			iStepSectionWork:=iStepSection;		(* set the actual section which is working *)
			IF ((iStepSection + (iStartSection - 1)) < iEndSection) THEN	(* check if the end section is active *)
				iStepSection:=iStepSection + 1;
			ELSE
				iStepSection:=5;	(* end section is reached-->go the displace procedure *)
			END_IF;
	(* plunge procedure *)
	5:		rActualPositionGrindFeedStart[5]:=rActualPositionGrindFeedEnd[iEndSection - (iStartSection - 1)];	(* set the new diameter of the section which will going to work *)
			rDistanceToWorkedTool:=rActualPositionGrindFeedStart[5] - rToolDiameterWithOffset;	(* check the distance to the end diameter, which will go to work *)
			rGrindingRelativePosition:=rDistanceToWorkedTool;
			IF (rActualPositionGrindFeedStart[5] = T_Geometry.arEndDiameter[iEndSection]) THEN
				axWorkEndSection[5]:=TRUE;		(* the end of this section is reached *)
			ELSE
				axWorkEndSection[5]:=FALSE;		(* the end of this section is not reached *)
			END_IF;
			rActualPositionGrindFeedEnd[5]:=rToolDiameterWithOffset;
			iStepSectionWork:=iStepSection;		(* set the actual section which is working *)
			iStepSection:=0;
END_CASE;
END_FUNCTION_BLOCK

(* POU PRG_VISU_LAYER5/FB_VISU/iFctGetEditParaList, ST *)
FUNCTION iFctGetEditParaList : INT
VAR_INPUT
	dwActualPage:DWORD;		(* activate page on the visualisation *)
	xMicroRodActive: BOOL;		(* choice of the machine MicroWire or MicroRod *)
	iSelectParaList:INT;			(* parameter list choiced on the QVis *)
	iSelectParaListTeachRot:INT;	(* parameter list choiced on the QVis for teach ToolRotation *)
END_VAR
VAR
	iTmpRetEditParaList: INT;
END_VAR
(****************************************************************************************************************************************************)
(***********          This Function check the state of the parameter level and give the number of the parameter list                ************)
(****************************************************************************************************************************************************)
iTmpRetEditParaList:=0;
CASE dwActualPage OF
	110:	IF xMicroRodActive THEN
			iTmpRetEditParaList:=111;
		ELSE
			iTmpRetEditParaList:=110;
		END_IF;
	120:	IF (iSelectParaList = 0) OR (iSelectParaList = 1) THEN
			IF xMicroRodActive THEN
				iTmpRetEditParaList:=123;
			ELSE
				iTmpRetEditParaList:=120;
			END_IF;
		END_IF;
		IF (iSelectParaList = 2) THEN
			iTmpRetEditParaList:=121;
		END_IF;
		IF (iSelectParaList = 3) THEN
			IF xMicroRodActive THEN
				iTmpRetEditParaList:=125;
			ELSE
				iTmpRetEditParaList:=122;
			END_IF;
		END_IF;
	130:	IF xMicroRodActive THEN
			iTmpRetEditParaList:=131;
		ELSE
			iTmpRetEditParaList:=130;
		END_IF;
	140:	iTmpRetEditParaList:=140;
	150:	iTmpRetEditParaList:=150;
	210:	IF (iSelectParaListTeachRot = 0) OR (iSelectParaListTeachRot = 1) THEN
			iTmpRetEditParaList:=210;
		END_IF;
		IF (iSelectParaListTeachRot = 2) THEN
			iTmpRetEditParaList:=211;
		END_IF;
		IF (iSelectParaListTeachRot = 3) THEN
			iTmpRetEditParaList:=212;
		END_IF;
	220:	iTmpRetEditParaList:=0;
	230:	iTmpRetEditParaList:=230;
	310:IF xMicroRodActive THEN
			iTmpRetEditParaList:=311;
		ELSE
			iTmpRetEditParaList:=310;
		END_IF;
	320:	iTmpRetEditParaList:=0;
	410:	iTmpRetEditParaList:=410;
	420:	iTmpRetEditParaList:=0;
	430:	iTmpRetEditParaList:=0;
END_CASE;
iFctGetEditParaList:=iTmpRetEditParaList;
END_FUNCTION

(* POU PRG_VISU_LAYER5/FB_VISU/iFctReturnConfMessage, ST *)
FUNCTION iFctReturnConfMessage : INT
VAR_INPUT
	iNumAction:INT;	(* number of called action on the visualisation *)
END_VAR
VAR
END_VAR
(****************************************************************************************************************************************************)
(***********                      This Function check the action on the visu and gives a correspond message number                     ************)
(****************************************************************************************************************************************************)
	CASE iNumAction OF
	(* Action exceeded Timeout *)
	-1:	iFctReturnConfMessage:=102;
	(* NovRAM, 'Parameter saved' with confirmation *)
	1005:	iFctReturnConfMessage:=1;
	(* NovRAM, 'Parameter saved' without confirmation *)
	1006:	iFctReturnConfMessage:=1;
	(* Reference machine done *)
	1110:	iFctReturnConfMessage:=23;
	(* Process machine done *)
	1150:	iFctReturnConfMessage:=21;
	(* Process station done *)
	1151..1153:	iFctReturnConfMessage:=22;
	(* change page, no message *)
	10001..10999:	iFctReturnConfMessage:=0;
	(* Info , 'Confirm action' *)
	ELSE	iFctReturnConfMessage:=2;
	END_CASE
END_FUNCTION

(* POU PRG_VISU_LAYER5/FB_VISU/xFctCtrleProfileName, ST *)
FUNCTION xFctCtrleProfileName : BOOL
VAR_INPUT
	sNewProfileName:STRING(30);		(* profile name to save *)
	ptrProfileList:POINTER TO ARRAY[1..csiMaxProfile] OF ST_PROFILE_ID;	(* list of the saved profil names *)
END_VAR
VAR
(* variable *)
	i: INT;
	sTmp:STRING;
	sTmp2:STRING;
END_VAR
(****************************************************************************************************************************************************)
(***********                                              This Function check the name of the profile if it is correct                                                     ************)
(****************************************************************************************************************************************************)
(* Init. function *)
	xFctCtrleProfileName:=FALSE;
	sTmp:=FCT_UPLOW_CASE(	xLowConvert:=TRUE,
							sInString:=sNewProfileName);

(* Search if name already exists *)
	FOR i:=1 TO csiMaxProfile DO
		sTmp2:=	FCT_UPLOW_CASE(	xLowConvert:=TRUE,
								sInString:=ptrProfileList^[i].sName);
		IF sTmp = sTmp2 AND sTmp2 <> '' THEN RETURN; END_IF
	END_FOR

(* Confirm function *)
	xFctCtrleProfileName:=TRUE;
END_FUNCTION

(* POU GENERAL/FCT_UPLOW_CASE, ST *)
FUNCTION FCT_UPLOW_CASE : STRING
VAR_INPUT
	xLowConvert:BOOL;			(* FALSE=conversion to up case, TRUE=conversion in low case *)
	sInString:STRING;				(* string with 80 character, which will be convert *)
END_VAR
VAR
(* variable *)
	sListUpCase:STRING:='ABCDEFGHIJKLMNOPQRSTUVWXYZ';
	sListLowCase:STRING:='abcdefghijklmnopqrstuvwxyz';
	i:INT;
(* Tmp *)
	sTmp:STRING;
	iTmp:INT;
END_VAR
(****************************************************************************************************************************************************)
(***********                                                      This function convert a String in up or low case                                                                ************)
(****************************************************************************************************************************************************)
(* Init. *)
	FCT_UPLOW_CASE:='';

(*Test string size*)
	IF LEN(sInString) < 1 OR LEN(sInString) > 255 THEN RETURN; END_IF

	IF xLowConvert THEN
	(* Conversion to low case *)
		FOR i:= 1 TO LEN(sInString) DO
			sTmp:=MID(sInString,1,i);
			iTmp:=FIND(sListUpCase,sTmp);
			IF iTmp > 0 THEN FCT_UPLOW_CASE:=CONCAT(FCT_UPLOW_CASE,MID(sListLowCase,1,iTmp));
				ELSE FCT_UPLOW_CASE:=CONCAT(FCT_UPLOW_CASE,sTmp); END_IF
		END_FOR
	(* Conversion to up case *)
	ELSE
		FOR i:= 1 TO LEN(sInString) DO
			sTmp:=MID(sInString,1,i);
			iTmp:=FIND(sListLowCase,sTmp);
			IF iTmp > 0 THEN FCT_UPLOW_CASE:=CONCAT(FCT_UPLOW_CASE,MID(sListUpCase,1,iTmp));
				ELSE FCT_UPLOW_CASE:=CONCAT(FCT_UPLOW_CASE,sTmp); END_IF
		END_FOR
	END_IF
END_FUNCTION

(* POU PRG_VISU_LAYER5/FB_VISU/iFctExistProfileName, ST *)
FUNCTION iFctExistProfileName : INT
VAR_INPUT
	sProfileName:STRING(30);											(* name of the profile, which will be saved *)
	ptrProfileList:POINTER TO ARRAY[1..csiMaxProfile] OF ST_PROFILE_ID;	(* list of profil names which are saved *)
END_VAR
VAR
	i:INT;
	sTmp:STRING;
	sTmp2:STRING;
END_VAR
(****************************************************************************************************************************************************)
(***********                                               This Function check if the name of the profile already exists                                              ************)
(****************************************************************************************************************************************************)
(* Init. function *)
	iFctExistProfileName:=0;
	sTmp:=FCT_UPLOW_CASE(	xLowConvert:=TRUE,
							sInString:=sProfileName);

(* Search if name already exists *)
	FOR i:=1 TO csiMaxProfile DO
		sTmp2:=	FCT_UPLOW_CASE(	xLowConvert:=TRUE,
								sInString:=ptrProfileList^[i].sName);
		IF sTmp = sTmp2 AND sTmp2 <> '' THEN iFctExistProfileName:=i; RETURN; END_IF
	END_FOR
END_FUNCTION

(* POU PRG_VISU_LAYER5/FB_VISU/rFctCalcMaxToolDiameter, ST *)
FUNCTION rFctCalcMaxToolDiameter : REAL
VAR_INPUT
	rDistanceD1:REAL;		(* distance d1 of the prisma *)
	rDistanceD2:REAL;		(* distance d2 of the prisma *)
	rAnglePrism:REAL;		(* angle of the prisma *)
END_VAR
VAR
	rTmp: REAL;
	rTmpMaxDia: REAL;
END_VAR
(****************************************************************************************************************************************************)
(***********                    This Function calculate the maximum of the tooldiameter in case of the settled prisma                      ************)
(****************************************************************************************************************************************************)
rTmp:=SIN((90 - rAnglePrism/2) * PI/180);
IF rTmp <> 0 THEN
	rTmpMaxDia:=rDistanceD1/rTmp;
ELSE
	rTmpMaxDia:=0;
END_IF;
rFctCalcMaxToolDiameter:=rTmpMaxDia;
END_FUNCTION

(* POU PRG_VISU_LAYER5/FB_VISU/rFctCalcMinToolDiameter, ST *)
FUNCTION rFctCalcMinToolDiameter : REAL
VAR_INPUT
	rDistanceD1:REAL;		(* distance d1 of the prisma *)
	rDistanceD2:REAL;		(* distance d2 of the prisma *)
	rAnglePrism:REAL;		(* angle of the prisma *)
	bStateInputPrisma:BYTE;	(* choice of selected prisma *)
END_VAR
VAR
	rTmp: REAL;
	rTmp1: REAL;
	rMinD1_1: REAL;
	rMinD1_2: REAL;
	rReturnValue: REAL;
END_VAR
(****************************************************************************************************************************************************)
(***********                    This Function calculate the minimum of the tooldiameter in case of the settled prisma                      ************)
(****************************************************************************************************************************************************)
rFctCalcMinToolDiameter:=0;
rTmp:=TAN((rAnglePrism/2)*PI/180);
rTmp1:=SIN((rAnglePrism/2)*PI/180);
IF (rTmp <> 0) AND (rTmp1 <> 0) THEN
	rMinD1_1:=rDistanceD1/(rTmp * (1 + 1/rTmp1));
END_IF;
rMinD1_2:=rDistanceD2;
IF (bStateInputPrisma = 0) OR (bStateInputPrisma = 1) THEN
	IF (rMinD1_1 >= rMinD1_2) THEN
		rReturnValue:=rMinD1_1;
	ELSE
		rReturnValue:=rMinD1_2;
	END_IF;
ELSE
	rReturnValue:=rMinD1_1;
END_IF;
rFctCalcMinToolDiameter:=rReturnValue;
END_FUNCTION

(* POU PRG_VISU_LAYER5/FB_VISU/rFctCalcPrismaFactor, ST *)
FUNCTION rFctCalcPrismaFactor : REAL
VAR_INPUT
	rAnglePrism:REAL;	(* angle of the prisma *)
END_VAR
VAR
	rFactorPrisma: REAL;
END_VAR
(****************************************************************************************************************************************************)
(***********     This Function calculate the correctur factor for the GrindFeeder Axis dependent of the settled prisma         ************)
(****************************************************************************************************************************************************)
rFctCalcPrismaFactor:=0.0;
rFactorPrisma:=(1 + SIN((rAnglePrism / 2.0) * PI/180)) / (2.0 * SIN((rAnglePrism / 2.0) * PI / 180.0));
(* Auf 5 Kommastellen runden *)
rFactorPrisma:=	STRING_TO_REAL(	LREAL_TO_FMTSTR(	in:=rFactorPrisma,
														iPrecision:=5,
														bRound:=TRUE));

rFctCalcPrismaFactor:=rFactorPrisma;
END_FUNCTION

(* POU PRG_VISU_LAYER5/FB_VISU/FB_CTRLEBUTTON, ST *)
FUNCTION_BLOCK FB_CTRLEBUTTON
VAR_INPUT
	xHWStart:BOOL;							(* external start button *)
	xHWStop:BOOL;							(* external stop button *)
	dwActualPage:DWORD;					(* active number page of the visualisation *)
	T_VisuQVis:ST_QVIS;						(* data structure of the visualisation *)
	T_ExchgParam:ST_QVIS_EXCHG_PARAM;	(* data structure of the visualisation *)
	IxSafetyCircuitOn1:BOOL;					(* state of current if it is on or off from the channel 1 *)
	IxSafetyCircuitOn2:BOOL;					(* state of current if it is on or off from the channel 2 *)
END_VAR
VAR_OUTPUT
END_VAR
VAR_IN_OUT
	T_StartButton: ST_BUTTON;				(* data structure of the control button start *)
	T_StopButton:ST_BUTTON;				(* data structure of the control button stop *)
END_VAR
VAR
(* Init. variable *)
	xFirstExecution:BOOL:=FALSE;
(* Variable *)
	iIndexActivPage:INT;
	dwOldActualPage:DWORD;
(* FB Mask *)
	xMaskPageBtStart:BOOL;
	xMaskPageBtStop:BOOL;
(* Trigger *)
	RisingEdgeSignalStartButton:R_TRIG;
	RisingEdgeStartState:R_TRIG;
	RisingEdgeCfgBtStart:R_TRIG;
	RisingEdgeSignalStopButton:R_TRIG;
	RisingEdgeFlagStopProcess:R_TRIG;
(* Tmp variable *)
	xTmp:BOOL;
END_VAR
(****************************************************************************************************************************************************)
(***********             This Functionblock manage the external start and stop butto, also for the lamp of this button                  ************)
(****************************************************************************************************************************************************)
(* First execution *)
	IF NOT xFirstExecution THEN
		dwOldActualPage:=16#FFFFFFFF;
		RisingEdgeSignalStartButton(CLK:=FALSE);
		RisingEdgeStartState(CLK:=FALSE);
		RisingEdgeCfgBtStart(CLK:=FALSE);
		RisingEdgeSignalStopButton(CLK:=FALSE);
		RisingEdgeFlagStopProcess(CLK:=FALSE);
		(* Set first execution *)
		xFirstExecution:=TRUE;
	END_IF

(* exit FB if Qvis inactiv *)
	IF NOT(T_VisuQVis.T_CtrleVisu.xQvis) THEN RETURN; END_IF
	IF (dwActualPage < 1) OR (dwActualPage > 999) THEN RETURN; END_IF;

(* Index Activ Page *)
	IF dwActualPage = 0 THEN iIndexActivPage:=1;
	ELSE iIndexActivPage:=T_VisuQVis.T_PageIndex[dwActualPage].iIndexConfigPage; END_IF

(* Start Button *)
	xMaskPageBtStart:=FALSE;
	CASE dwActualPage OF
	(* Auto Geometry page *)
	10:	xTmp:=TRUE;
		IF xTmp AND (NOT(IxSafetyCircuitOn1) OR NOT(IxSafetyCircuitOn2)) THEN
			xTmp:=FALSE;	(* Energieversorgung muss eingeschaltet sein *)
		END_IF;
		IF xTmp AND ((T_ExchgParam.T_SafetyCtrl.bStateMessageError <> 0) OR (T_ExchgParam.T_SafetyCtrl.bStateMessageInfo <> 0)) THEN
			xTmp:=FALSE;
		END_IF;
		IF (T_ExchgParam.T_Visu.T_Message.iState = 401) OR (T_ExchgParam.T_Visu.T_Message.iState = 118) OR (T_ExchgParam.T_Visu.T_Message.iState = 119) OR (T_ExchgParam.T_Visu.T_Message.iState = 108) THEN
			xTmp:=FALSE;
		END_IF;
		(* copy state *)
		xMaskPageBtStart:=xTmp;
	(* Auto Groove page *)
	20:	xTmp:=TRUE;
		IF xTmp AND (NOT(IxSafetyCircuitOn1) OR NOT(IxSafetyCircuitOn2)) THEN
			xTmp:=FALSE;	(* Energieversorgung muss eingeschaltet sein *)
		END_IF;
		IF xTmp AND ((T_ExchgParam.T_SafetyCtrl.bStateMessageError <> 0) OR (T_ExchgParam.T_SafetyCtrl.bStateMessageInfo <> 0)) THEN
			xTmp:=FALSE;
		END_IF;
		IF (T_ExchgParam.T_Visu.T_Message.iState = 401) OR (T_ExchgParam.T_Visu.T_Message.iState = 118) OR (T_ExchgParam.T_Visu.T_Message.iState = 119) OR (T_ExchgParam.T_Visu.T_Message.iState = 108) THEN
			xTmp:=FALSE;
		END_IF;
		(* copy state *)
		xMaskPageBtStart:=xTmp;
	(* Reference page *)
	30:	xTmp:=TRUE;
		IF xTmp AND (NOT(IxSafetyCircuitOn1) OR NOT(IxSafetyCircuitOn2)) THEN
			xTmp:=FALSE;	(* Energieversorgung muss eingeschaltet sein *)
		END_IF;
		IF xTmp AND ((T_ExchgParam.T_SafetyCtrl.bStateMessageError <> 0) OR (T_ExchgParam.T_SafetyCtrl.bStateMessageInfo <> 0)) THEN
			xTmp:=FALSE;
		END_IF;
		IF (T_ExchgParam.T_Visu.T_Message.iState = 401) OR (T_ExchgParam.T_Visu.T_Message.iState = 118) OR (T_ExchgParam.T_Visu.T_Message.iState = 119) THEN
			xTmp:=FALSE;
		END_IF;
		IF (T_ExchgParam.T_StationCommon.iConfigMachineType = 1) THEN
			xTmp:=FALSE;
		END_IF;
		(* copy state *)
		xMaskPageBtStart:=xTmp;
	(* Tool Calibration page *)
	110:	xTmp:=TRUE;
		IF xTmp AND (NOT(IxSafetyCircuitOn1) OR NOT(IxSafetyCircuitOn2)) THEN
			xTmp:=FALSE;	(* Energieversorgung muss eingeschaltet sein *)
		END_IF;
		IF xTmp AND ((T_ExchgParam.T_SafetyCtrl.bStateMessageError <> 0) OR (T_ExchgParam.T_SafetyCtrl.bStateMessageInfo <> 0)) THEN
			xTmp:=FALSE;
		END_IF;
		IF (T_ExchgParam.T_Visu.T_Message.iState = 401) OR (T_ExchgParam.T_Visu.T_Message.iState = 118) OR (T_ExchgParam.T_Visu.T_Message.iState = 119) OR
		     (T_ExchgParam.T_Visu.T_Message.iState = 108) THEN
			xTmp:=FALSE;
		END_IF;
		IF ((T_ExchgParam.T_Machine.T_Process.wState AND 16#6) = 16#2) THEN
			xTmp:=FALSE;
		END_IF;
		IF T_ExchgParam.T_FunctionCommon.xOpenOverlayMeasureInput OR T_ExchgParam.T_FunctionCommon.xOpenOverlaySetGrindPlunge THEN
			xTmp:=FALSE;
		END_IF;
		(* copy state *)
		xMaskPageBtStart:=xTmp;
	(* Teach-in Tool Rotation page *)
	210:	xTmp:=	((T_ExchgParam.T_StationCommon.bStateMachine AND 16#7) = 16#1);
		IF xTmp AND (NOT(IxSafetyCircuitOn1) OR NOT(IxSafetyCircuitOn2)) THEN
			xTmp:=FALSE;	(* Energieversorgung muss eingeschaltet sein *)
		END_IF;
		IF xTmp AND ((T_ExchgParam.T_SafetyCtrl.bStateMessageError <> 0) OR (T_ExchgParam.T_SafetyCtrl.bStateMessageInfo <> 0)) THEN
			xTmp:=FALSE;
		END_IF;
		IF (T_ExchgParam.T_Visu.T_Message.iState = 401) OR (T_ExchgParam.T_Visu.T_Message.iState = 118) OR (T_ExchgParam.T_Visu.T_Message.iState = 119) OR
		     (T_ExchgParam.T_Visu.T_Message.iState = 101) THEN
			xTmp:=FALSE;
		END_IF;
		IF (T_ExchgParam.T_TeachIn.iSelectAxisToolRotation = 1) AND xTmp THEN
			IF ((T_ExchgParam.T_StationCommon.bStateAxisReelLeft AND 16#2) = 16#2) THEN
				xTmp:=FALSE;
			END_IF;
		END_IF;
		IF (T_ExchgParam.T_TeachIn.iSelectAxisToolRotation = 2) AND xTmp THEN
			IF ((T_ExchgParam.T_StationCommon.bStateAxisReelCenter AND 16#2) = 16#2) THEN
				xTmp:=FALSE;
			END_IF;
		END_IF;
		IF (T_ExchgParam.T_TeachIn.iSelectAxisToolRotation = 3) AND xTmp THEN
			IF ((T_ExchgParam.T_StationCommon.bStateAxisReelRight AND 16#2) = 16#2) THEN
				xTmp:=FALSE;
			END_IF;
		END_IF;
		(* copy state *)
		xMaskPageBtStart:=xTmp;
	(* Tool Torque page *)
	220:	xTmp:=	((T_ExchgParam.T_StationCommon.bStateMachine AND 16#7) = 16#1);
		IF xTmp AND (NOT(IxSafetyCircuitOn1) OR NOT(IxSafetyCircuitOn2)) THEN
			xTmp:=FALSE;	(* Energieversorgung muss eingeschaltet sein *)
		END_IF;
		IF xTmp AND ((T_ExchgParam.T_SafetyCtrl.bStateMessageError <> 0) OR (T_ExchgParam.T_SafetyCtrl.bStateMessageInfo <> 0)) THEN
			xTmp:=FALSE;
		END_IF;
		IF (T_ExchgParam.T_Visu.T_Message.iState = 401) OR (T_ExchgParam.T_Visu.T_Message.iState = 118) OR (T_ExchgParam.T_Visu.T_Message.iState = 119) OR
		     (T_ExchgParam.T_Visu.T_Message.iState = 101) THEN
			xTmp:=FALSE;
		END_IF;
		IF ((T_ExchgParam.T_StationCommon.bStateAxisReelLeft AND 16#2) = 16#2) THEN
			xTmp:=FALSE;
		END_IF;
		(* copy state *)
		xMaskPageBtStart:=xTmp;
	(* Teach-in Tool Feeder page *)
	310:	xTmp:=	xTmp:=	((T_ExchgParam.T_StationCommon.bStateMachine AND 16#7) = 16#1);
		IF xTmp AND (NOT(IxSafetyCircuitOn1) OR NOT(IxSafetyCircuitOn2)) THEN
			xTmp:=FALSE;	(* Energieversorgung muss eingeschaltet sein *)
		END_IF;
		IF xTmp AND ((T_ExchgParam.T_SafetyCtrl.bStateMessageError <> 0) OR (T_ExchgParam.T_SafetyCtrl.bStateMessageInfo <> 0)) THEN
			xTmp:=FALSE;
		END_IF;
		IF (T_ExchgParam.T_Visu.T_Message.iState = 401) OR (T_ExchgParam.T_Visu.T_Message.iState = 118) OR (T_ExchgParam.T_Visu.T_Message.iState = 119) OR
		     (T_ExchgParam.T_Visu.T_Message.iState = 101) OR (T_ExchgParam.T_Visu.T_Message.iState = 18) THEN
			xTmp:=FALSE;
		END_IF;
		IF (T_ExchgParam.T_TeachIn.iSelectAxisWireFeeder = 1) AND xTmp THEN
			IF ((T_ExchgParam.T_StationCommon.bStateAxisWireFeeder AND 16#2) = 16#2) THEN
				xTmp:=FALSE;
			END_IF;
		END_IF;
		(* copy state *)
		xMaskPageBtStart:=xTmp;
	(* Teach-in Tool Feeder page *)
	330:	xTmp:=	xTmp:=	((T_ExchgParam.T_StationCommon.bStateMachine AND 16#7) = 16#1);
		IF xTmp AND (NOT(IxSafetyCircuitOn1) OR NOT(IxSafetyCircuitOn2)) THEN
			xTmp:=FALSE;	(* Energieversorgung muss eingeschaltet sein *)
		END_IF;
		IF xTmp AND ((T_ExchgParam.T_SafetyCtrl.bStateMessageError <> 0) OR (T_ExchgParam.T_SafetyCtrl.bStateMessageInfo <> 0)) THEN
			xTmp:=FALSE;
		END_IF;
		IF (T_ExchgParam.T_Visu.T_Message.iState = 401) OR (T_ExchgParam.T_Visu.T_Message.iState = 118) OR (T_ExchgParam.T_Visu.T_Message.iState = 119) OR
		     (T_ExchgParam.T_Visu.T_Message.iState = 101) OR (T_ExchgParam.T_Visu.T_Message.iState = 18) THEN
			xTmp:=FALSE;
		END_IF;
		IF (T_ExchgParam.T_TeachIn.iSelectAxisWireFeeder = 1) AND xTmp THEN
			IF ((T_ExchgParam.T_StationCommon.bStateAxisWireFeeder AND 16#2) = 16#2) THEN
				xTmp:=FALSE;
			END_IF;
		END_IF;
		(* copy state *)
		xMaskPageBtStart:=xTmp;
	(* Teach-in Grind Feeder page *)
	410:	xTmp:=	xTmp:=	((T_ExchgParam.T_StationCommon.bStateMachine AND 16#7) = 16#1);
		IF xTmp AND (NOT(IxSafetyCircuitOn1) OR NOT(IxSafetyCircuitOn2)) THEN
			xTmp:=FALSE;	(* Energieversorgung muss eingeschaltet sein *)
		END_IF;
		IF xTmp AND ((T_ExchgParam.T_SafetyCtrl.bStateMessageError <> 0) OR (T_ExchgParam.T_SafetyCtrl.bStateMessageInfo <> 0)) THEN
			xTmp:=FALSE;
		END_IF;
		IF (T_ExchgParam.T_Visu.T_Message.iState = 401) OR (T_ExchgParam.T_Visu.T_Message.iState = 118) OR (T_ExchgParam.T_Visu.T_Message.iState = 119) OR
		     (T_ExchgParam.T_Visu.T_Message.iState = 101) THEN
			xTmp:=FALSE;
		END_IF;
		IF (T_ExchgParam.T_TeachIn.iSelectAxisGrind = 1) AND xTmp THEN
			IF ((T_ExchgParam.T_StationCommon.bStateAxisGrind AND 16#2) = 16#2) THEN
				xTmp:=FALSE;
			END_IF;
		END_IF;
		(* copy state *)
		xMaskPageBtStart:=xTmp;
	END_CASE

	(* Set state button start *)
	RisingEdgeSignalStartButton(CLK:=xHWStart);
	IF RisingEdgeSignalStartButton.Q THEN T_StartButton.xInputState:=TRUE; ELSE T_StartButton.xInputState:=FALSE; END_IF
	T_StartButton.xInputState:=T_StartButton.xInputState AND T_VisuQVis.T_ConfigPage[iIndexActivPage].xMaskBtStart;

	(* if page change => init. trigger *)
	IF dwActualPage <> dwOldActualPage THEN
		RisingEdgeStartState(CLK:=FALSE);
		RisingEdgeCfgBtStart(CLK:=FALSE);
		(* save value *)
		dwOldActualPage:=dwActualPage;
	END_IF

	(* Led off if action is starting *)
	RisingEdgeStartState(CLK:=T_StartButton.xInputState);
	IF RisingEdgeStartState.Q THEN T_StartButton.xLedState:=FALSE; END_IF
	RisingEdgeCfgBtStart(CLK:=xMaskPageBtStart);
	IF RisingEdgeCfgBtStart.Q THEN T_StartButton.xLedState:=TRUE; END_IF
	T_StartButton.xLedState:=T_StartButton.xLedState AND T_VisuQVis.T_ConfigPage[iIndexActivPage].xMaskBtStart;

	(* set page mask *)
	T_StartButton.xInputState:=T_StartButton.xInputState AND xMaskPageBtStart;
	T_StartButton.xLedState:=T_StartButton.xLedState AND xMaskPageBtStart;

(* Stop Button *)
	xMaskPageBtStop:=FALSE;
	RisingEdgeSignalStopButton(CLK:=xHWStop);
	IF RisingEdgeSignalStopButton.Q THEN T_StopButton.xInputState:=TRUE; ELSE T_StopButton.xInputState:=FALSE; END_IF
	T_StopButton.xInputState:=T_StopButton.xInputState AND T_VisuQVis.T_ConfigPage[iIndexActivPage].xMaskBtStop;
	T_StopButton.xLedState:=T_VisuQVis.T_ConfigPage[iIndexActivPage].xMaskBtStop;

	(* if machine process inactiv => set mask inactiv *)
	IF dwActualPage > 0 THEN
		IF (T_ExchgParam.T_Machine.T_Process.wState AND 16#14) = 16#0 THEN
		(* process activ and no error *)
			IF (T_ExchgParam.T_Machine.T_Process.wState AND 16#80) = 16#0 THEN xMaskPageBtStop:=TRUE; ELSE xMaskPageBtStop:=FALSE; END_IF
		ELSIF ((dwActualPage = 210) OR (dwActualPage = 310) OR (dwActualPage = 410)) THEN
			(* Achse muss Aktiv sein, Stationsendflag muss gesetzt sein, Prozessendflag muss gesetzt sein *)
			IF ((T_ExchgParam.T_StationCommon.bStateMachine AND 16#7) = 16#3) AND ((T_ExchgParam.T_Machine.T_Process.wState AND 16#2) = 16#0) THEN
				xMaskPageBtStop:=TRUE;
			END_IF;
			(* Achse darf nicht Aktiv sein, Stationsendflag muss gesetzt sein,  Prozessendflag muss gesetzt sein *)
			IF ((T_ExchgParam.T_StationCommon.bStateMachine AND 16#7) = 16#1) AND ((T_ExchgParam.T_Machine.T_Process.wState AND 16#2) = 16#0) THEN
				xMaskPageBtStop:=FALSE;
				IF (T_ExchgParam.T_TeachIn.iSelectAxisToolRotation = 1) AND (dwActualPage = 210) THEN
					IF ((T_ExchgParam.T_StationCommon.bStateAxisReelLeft AND 16#2) = 16#2) THEN
						xMaskPageBtStop:=TRUE;
					END_IF;
				END_IF;
				IF (T_ExchgParam.T_TeachIn.iSelectAxisToolRotation = 2) AND (dwActualPage = 210) THEN
					IF ((T_ExchgParam.T_StationCommon.bStateAxisReelCenter AND 16#2) = 16#2) THEN
						xMaskPageBtStop:=TRUE;
					END_IF;
				END_IF;
				IF (T_ExchgParam.T_TeachIn.iSelectAxisToolRotation = 3) AND (dwActualPage = 210) THEN
					IF ((T_ExchgParam.T_StationCommon.bStateAxisReelRight AND 16#2) = 16#2) THEN
						xMaskPageBtStop:=TRUE;
					END_IF;
				END_IF;
				IF (T_ExchgParam.T_TeachIn.iSelectAxisWireFeeder = 1) AND (dwActualPage = 310) THEN
					IF ((T_ExchgParam.T_StationCommon.bStateAxisWireFeeder AND 16#2) = 16#2) THEN
						xMaskPageBtStop:=TRUE;
					END_IF;
				END_IF;
				IF (T_ExchgParam.T_TeachIn.iSelectAxisGrind = 1) AND (dwActualPage = 410) THEN
					IF ((T_ExchgParam.T_StationCommon.bStateAxisGrind AND 16#2) = 16#2) THEN
						xMaskPageBtStop:=TRUE;
					END_IF;
				END_IF;
			END_IF;
			IF (T_VisuQVis.T_CtrleAction.iFunction = 301) AND NOT(T_VisuQVis.T_CtrleAction.xDone) THEN
				xMaskPageBtStop:=FALSE;
			END_IF;
		ELSIF (dwActualPage = 220) THEN
			(* Achse muss Aktiv sein, Stationsendflag muss gesetzt sein, Prozessendflag muss gesetzt sein *)
			xMaskPageBtStop:=FALSE;
			IF ((T_ExchgParam.T_StationCommon.bStateAxisReelLeft AND 16#2) = 16#2) THEN
				xMaskPageBtStop:=TRUE;
			END_IF;
			IF (T_VisuQVis.T_CtrleAction.iFunction = 403) AND NOT(T_VisuQVis.T_CtrleAction.xDone) THEN
				xMaskPageBtStop:=FALSE;
			END_IF;
		(* process inactiv *)
		ELSE xMaskPageBtStop:=FALSE; END_IF
		IF (T_ExchgParam.T_Visu.T_Message.iState = 401) OR (T_ExchgParam.T_Visu.T_Message.iState = 118) OR (T_ExchgParam.T_Visu.T_Message.iState = 119) THEN
			xMaskPageBtStop:=FALSE;
		END_IF;
		IF NOT(IxSafetyCircuitOn1) OR NOT(IxSafetyCircuitOn2) THEN
			xMaskPageBtStop:=FALSE;
		END_IF;
	END_IF

	(* set page mask *)
	T_StopButton.xInputState:=T_StopButton.xInputState AND xMaskPageBtStop;
	T_StopButton.xLedState:=T_StopButton.xLedState AND xMaskPageBtStop;
END_FUNCTION_BLOCK

(* POU PRG_PROCESS_LAYER4/PRG_PROCESS, FBD *)
PROGRAM PRG_PROCESS
VAR
	FBProcess: FB_PROCESS;
	xReady: BOOL;
	xEnd: BOOL;
	xStop: BOOL;
	xReferenced: BOOL;
	xError: BOOL;
	iErrorNr: DINT;
	iFunctionNr: INT;
END_VAR
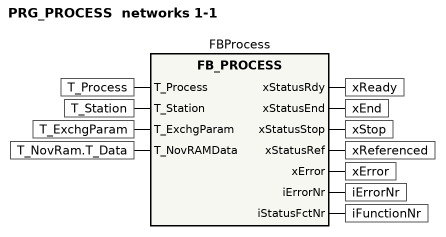
_FBD_ (* Function Block Diagram *)
NETWORK 1 (* PROCESS LEVEL-->LAYER 4 *)
	FBProcess:FB_PROCESS(T_Process: T_Process, T_Station: T_Station, T_ExchgParam: T_ExchgParam, T_NovRAMData: T_NovRam.T_Data, xStatusEnd => xEnd, xStatusStop => xStop, xStatusRef => xReferenced, xError => xError, iErrorNr => iErrorNr, iStatusFctNr => iFunctionNr) => xReady
_END_FBD_
(* the same logic as Structured Text *)
(* Network 1: PROCESS LEVEL-->LAYER 4 *)
FBProcess(T_Process := T_Process, T_Station := T_Station, T_ExchgParam := T_ExchgParam, T_NovRAMData := T_NovRam.T_Data);
xEnd := FBProcess.xStatusEnd;
xStop := FBProcess.xStatusStop;
xReferenced := FBProcess.xStatusRef;
xError := FBProcess.xError;
iErrorNr := FBProcess.iErrorNr;
iFunctionNr := FBProcess.iStatusFctNr;
xReady := FBProcess.xStatusRdy;
END_PROGRAM

(* POU PRG_PROCESS_LAYER4/FB_PROCESS/FB_PROCESS, ST *)
FUNCTION_BLOCK FB_PROCESS
VAR_INPUT
END_VAR
VAR_IN_OUT
	T_Process : ST_PROCESS;				(* data structure of the processlevel *)
	T_Station : ST_STATION;					(* data structure of the stationlevel *)
	T_ExchgParam:ST_QVIS_EXCHG_PARAM;	(* data structure of the visualisation *)
	T_NovRAMData:ST_DATA_RETAIN;		(* data structure of the NovRam *)
END_VAR
VAR_OUTPUT
	xStatusRdy : BOOL := FALSE;				(* state of the processlevel if it is ready or not *)
	xStatusEnd : BOOL := FALSE;				(* state of the processlevel if a process is active or not *)
	xStatusStop : BOOL := FALSE;				(* state of the processlevel if a process will be stopped *)
	xStatusRef : BOOL := FALSE;				(* state of the processlevel if the machine is referenced *)
	xError : BOOL := FALSE;					(* state of the processlevel if the machine has an error *)
	iErrorNr : DINT :=0;							(* state of the processlevel if the machine has an error, in this case it will give the errornumber *)
	iStatusFctNr : INT := 0;						(* state of the processlevel, which process is active *)
END_VAR
VAR
	xStartFunction: BOOL;
	xSetEnd: BOOL;
	iPrcFunctionNr: INT;
	xProcessError: BOOL;
	xInitError: BOOL;
	xTmpStart: BOOL;
	xInitStart: BOOL;
	xInitStop: BOOL;
	xTmpStopFunction: BOOL;
	xDisable: BOOL;
	xResetRef: BOOL;
	xInitStopCycle: BOOL;
	xTmpStopCycleFunction: BOOL;
(* end modif test torque *)
	FBErrorMessage : FB_ErrorMessage;
	FBPrcMachineReference: FB_PrcMachineReference;
	FBPrcAutoGeometry: FB_PrcAutoGeometry;
	diTmpErrorNr: DINT;
	xResetAutoGeometry: BOOL;
	FBPrcAutoGroove: FB_PrcAutoGroove;
	xResetAutoGroove: BOOL;
	FBPrcToolCalibration: FB_PrcToolCalibration;
	xResetToolCalibration: BOOL;
END_VAR
(****************************************************************************************************************************************************)
(***********                                            This Functionblock manage all the machine process                                                             ************)
(****************************************************************************************************************************************************)
IF NOT(T_Process.xEnable) THEN
	T_Process.xRdy:=FALSE;
	xDisable:=TRUE;
	RETURN;
ELSE
	IF xDisable THEN
		T_Process.xRdy:=TRUE;
		xDisable:=FALSE;
		xSetEnd:=TRUE;
	END_IF;
END_IF;
(******************************************************************************************************************************************)
(****************************				                  Status Part                                                            *****************************)
(******************************************************************************************************************************************)
xStatusRdy:=T_Process.xRdy;
xStatusEnd:=T_Process.xEnd;
xStatusRef:=T_Station.TControl.xReferenced;
T_Process.xReferenced:=xStatusRef;
xError:=T_Process.xError;
iStatusFctNr:=iPrcFunctionNr;
(******************************************************************************************************************************************)
(****************************				         Error Controlling Part                                                  *****************************)
(******************************************************************************************************************************************)
IF xProcessError OR (T_Process.TFctProcess.xError AND T_Process.xRdy AND NOT(xSetEnd)) THEN
	IF NOT(xInitError) THEN
		xInitError:=TRUE;
		xProcessError:=TRUE;
		T_Process.TFctProcess.xQuitErr:=TRUE;
		T_Process.xProcessHold:=FALSE;
		diTmpErrorNr:=T_Process.TFctProcess.diErrorNr;
	END_IF;
	IF NOT(T_Process.TFctProcess.xQuitErr) AND T_Process.TFctProcess.xEnd AND (T_Process.diErrorNr = 0)THEN
		FBErrorMessage(	diErrorNr:=diTmpErrorNr,
						T_ErrorList:=T_ErrorList);
		T_ExchgParam.T_Visu.T_Message.sDynamicTextEnglish:=FBErrorMessage.sErrorTextEnglish;
		T_ExchgParam.T_Visu.T_Message.sDynamicTextDeutsch:=FBErrorMessage.sErrorTextDeutsch;
		T_ExchgParam.T_Visu.T_Message.sDynamicTextFrancais:=FBErrorMessage.sErrorTextFrancais;
		T_Process.diErrorNr:=diTmpErrorNr;
		T_Process.xError:=TRUE;
	END_IF;
	IF T_Process.xQuitError AND NOT(T_Process.TFctProcess.xQuitErr) THEN
		T_Process.xProcessHold:=FALSE;
		T_ExchgParam.T_Visu.T_Message.sDynamicTextEnglish:='';
		T_ExchgParam.T_Visu.T_Message.sDynamicTextDeutsch:='';
		T_ExchgParam.T_Visu.T_Message.sDynamicTextFrancais:='';
		xInitError:=FALSE;
		T_Process.xQuitError:=FALSE;
		xSetEnd:=TRUE;
	END_IF;
END_IF;
(******************************************************************************************************************************************)
(****************************				         Main Controlling Part                                                  *****************************)
(******************************************************************************************************************************************)
IF (T_Process.xStart OR xTmpStart) AND T_Process.xRdy AND NOT(xSetEnd) THEN
	IF NOT(xInitStart) THEN
		xInitStart:=TRUE;
		xTmpStart:=TRUE;
		T_Process.xStop:=FALSE;
		T_Process.xStopCycle:=FALSE;
		T_Process.xStart:=FALSE;
		T_Process.xEnd:=FALSE;
		T_Process.xProcessHold:=FALSE;
		T_Process.TFctProcess.xStart:=TRUE;
		xStartFunction:=TRUE;
		iPrcFunctionNr:=T_Process.iFunctNr;
	END_IF;
	IF T_Process.xAbord AND (T_Process.xStopCycle OR T_Process.xStop) THEN
		T_Process.xStopCycle:=T_Process.xStop:=FALSE;		(* Prozess ist am abbrechen, diese Flag können nicht mehr berücksichtigt werden *)
	END_IF;
	IF T_Process.xStopCycle THEN
		IF NOT(xInitStopCycle) THEN
			xInitStopCycle:=TRUE;
			T_Process.TFctProcess.xStopCycle:=TRUE;
		END_IF;
		IF NOT(T_Process.TFctProcess.xStopCycle) AND T_Process.TFctProcess.xProcessHold THEN
			xInitStopCycle:=FALSE;
			T_Process.xStopCycle:=FALSE;
			T_Process.xProcessHold:=TRUE;
			xTmpStopCycleFunction:=TRUE;
		END_IF;
		IF NOT(T_Process.TFctProcess.xStopCycle) AND NOT(T_Process.TFctProcess.xProcessHold) THEN
			xInitStopCycle:=FALSE;
			T_Process.xStopCycle:=FALSE;
			T_Process.xProcessHold:=FALSE;
			xTmpStopCycleFunction:=FALSE;
		END_IF;
	END_IF;
	IF T_Process.xStop THEN
		IF NOT(xInitStop) THEN
			xInitStop:=TRUE;
			T_Process.TFctProcess.xStop:=TRUE;
		END_IF;
		IF NOT(T_Process.TFctProcess.xStop) AND T_Process.TFctProcess.xProcessHold THEN
			xInitStop:=FALSE;
			T_Process.xProcessHold:=TRUE;
			T_Process.xStop:=FALSE;
			xTmpStopFunction:=TRUE;
		END_IF;
		IF NOT(T_Process.TFctProcess.xStop) AND NOT(T_Process.TFctProcess.xProcessHold) THEN
			xInitStop:=FALSE;
			T_Process.xStop:=FALSE;
			T_Process.xProcessHold:=FALSE;
			xTmpStopFunction:=FALSE;
		END_IF;
	END_IF;
	IF T_Process.xStart AND (xTmpStopFunction OR xTmpStopCycleFunction) AND NOT(T_Process.xAbord) THEN
		T_Process.xStart:=T_Process.xProcessHold:=FALSE;
		xTmpStopFunction:=FALSE;
		xTmpStopCycleFunction:=FALSE;
		T_Process.TFctProcess.xStart:=TRUE;
	END_IF;
	IF T_Process.xAbord AND (xTmpStopFunction OR xTmpStopCycleFunction) THEN
		T_Process.xProcessHold:=FALSE;
		T_Process.xStart:=FALSE;
		xTmpStopFunction:=FALSE;
		xTmpStopCycleFunction:=FALSE;
		T_Process.TFctProcess.xAbord:=TRUE;
	END_IF;
	IF NOT(T_Process.TFctProcess.xStart) AND T_Process.TFctProcess.xEnd AND NOT(xProcessError) THEN
		xTmpStart:=FALSE;
		xInitStart:=FALSE;
		xSetEnd:=TRUE;
	END_IF;
END_IF;
(******************************************************************************************************************************************)
(****************************				              Funktionen                                                               *****************************)
(******************************************************************************************************************************************)
IF xStartFunction AND NOT(xSetEnd) THEN
	IF (iPrcFunctionNr = 10) THEN
	(* Process AutoGeometry *)
		FBPrcAutoGeometry(	xMicroRodActive:=(T_NovRAMData.T_Standard.T_MachineConfig.iConfigMachineType = 2),
							xBeckhoffDriveActive:=(T_NovRAMData.T_Standard.T_MachineConfig.iConfigAxisType = 2),
							xStart:=T_Process.TFctProcess.xStart ,
							xStop:=T_Process.TFctProcess.xStop ,
							xStopCycle:=T_Process.TFctProcess.xStopCycle,
							xQuitErr:=T_Process.TFctProcess.xQuitErr ,
							xAbord:=T_Process.TFctProcess.xAbord ,
							T_Station:= T_Station,
							T_Process:= T_Process,
							xReset:= xResetAutoGeometry,
							T_ExchgParam:= T_ExchgParam,
							T_NovRAMData:=T_NovRAMData,
							xEnd=>T_Process.TFctProcess.xEnd ,
							xError=>T_Process.TFctProcess.xError ,
							diErrorNr=>T_Process.TFctProcess.diErrorNr);
	END_IF;
	IF (iPrcFunctionNr = 20) THEN
	(* Process AutoGroove *)
		FBPrcAutoGroove(	xMicroRodActive:=(T_NovRAMData.T_Standard.T_MachineConfig.iConfigMachineType = 2),
							xBeckhoffDriveActive:=(T_NovRAMData.T_Standard.T_MachineConfig.iConfigAxisType = 2),
							xStart:=T_Process.TFctProcess.xStart ,
							xStop:=T_Process.TFctProcess.xStop ,
							xQuitErr:=T_Process.TFctProcess.xQuitErr ,
							xAbord:=T_Process.TFctProcess.xAbord ,
							T_Station:= T_Station,
							T_Process:= T_Process,
							xReset:= xResetAutoGroove,
							T_ExchgParam:= T_ExchgParam,
							xDoNotMoveGrindPosition:=T_NovRAMData.T_ProcessImageData.T_AutoGroovePara.xBlockGrindFeeder,
							xPlungeActive:=T_NovRAMData.T_ProcessImageData.T_AutoGroovePara.xPlungeActivationGroove,
							T_NovRAMData:=T_NovRAMData,
							xEnd=>T_Process.TFctProcess.xEnd ,
							xError=>T_Process.TFctProcess.xError ,
							diErrorNr=>T_Process.TFctProcess.diErrorNr);
	END_IF;
	IF (iPrcFunctionNr = 30) THEN
	(* Process Machine Reference *)
		FBPrcMachineReference(	xMicroRodActive:=(T_NovRAMData.T_Standard.T_MachineConfig.iConfigMachineType = 2),
								xBeckhoffDriveActive:=(T_NovRAMData.T_Standard.T_MachineConfig.iConfigAxisType = 2),
								xStart:=T_Process.TFctProcess.xStart ,
								xStop:=T_Process.TFctProcess.xStop ,
								xQuitErr:=T_Process.TFctProcess.xQuitErr ,
								xAbord:=T_Process.TFctProcess.xAbord ,
								T_Station:= T_Station,
								T_Process:= T_Process,
								xReset:= xResetRef,
								T_ExchgParam:= T_ExchgParam,
								T_NovRAMData:=T_NovRAMData,
								xEnd=>T_Process.TFctProcess.xEnd ,
								xError=>T_Process.TFctProcess.xError ,
								diErrorNr=>T_Process.TFctProcess.diErrorNr);
	END_IF;
	IF (iPrcFunctionNr = 40) THEN
	(* Process ToolCalibration *)
		FBPrcToolCalibration(	xMicroRodActive:=(T_NovRAMData.T_Standard.T_MachineConfig.iConfigMachineType = 2),
							xBeckhoffDriveActive:=(T_NovRAMData.T_Standard.T_MachineConfig.iConfigAxisType = 2),
							xStart:=T_Process.TFctProcess.xStart ,
							xStop:=T_Process.TFctProcess.xStop ,
							xQuitErr:=T_Process.TFctProcess.xQuitErr ,
							xAbord:=T_Process.TFctProcess.xAbord ,
							T_Station:= T_Station,
							T_Process:= T_Process,
							xReset:= xResetAutoGeometry,
							T_ExchgParam:= T_ExchgParam,
							T_NovRAMData:=T_NovRAMData,
							xEnd=>T_Process.TFctProcess.xEnd ,
							xError=>T_Process.TFctProcess.xError ,
							diErrorNr=>T_Process.TFctProcess.diErrorNr);
	END_IF;
END_IF;
(******************************************************************************************************************************************)
(****************************				         Init / Reset Hardware                                                 *****************************)
(******************************************************************************************************************************************)
IF xSetEnd THEN
	xStartFunction:=FALSE;
	xProcessError:=FALSE;
	xInitError:=FALSE;
	xInitStart:=FALSE;
	xInitStop:=FALSE;
	xSetEnd:=FALSE;
	xTmpStart:=FALSE;
	T_Process.xEnd:=TRUE;
	T_Process.xStart:=FALSE;
	T_Process.xStop:=FALSE;
	T_Process.xError:=FALSE;
	T_Process.diErrorNr:=0;
	T_Process.xAbord:=FALSE;
	T_Process.xQuitError:=FALSE;
	T_Process.wStatus:=0;
	T_Process.xAbord:=FALSE;
	T_Process.xStopCycle:=FALSE;
	T_Process.xProcessHold:=FALSE;
	xResetRef:=TRUE;
	FBPrcMachineReference(	xStart:=T_Process.TFctProcess.xStart ,
							xStop:=T_Process.TFctProcess.xStop ,
							xQuitErr:=T_Process.TFctProcess.xQuitErr ,
							xAbord:=T_Process.TFctProcess.xAbord ,
							T_Station:= T_Station,
							T_Process:= T_Process,
							xReset:= xResetRef,
							T_ExchgParam:= T_ExchgParam,
							xEnd=>T_Process.TFctProcess.xEnd ,
							xError=>T_Process.TFctProcess.xError ,
							diErrorNr=>T_Process.TFctProcess.diErrorNr);
	xResetAutoGeometry:=TRUE;
	FBPrcAutoGeometry(	xMicroRodActive:=(T_NovRAMData.T_Standard.T_MachineConfig.iConfigMachineType = 2),
						xBeckhoffDriveActive:=(T_NovRAMData.T_Standard.T_MachineConfig.iConfigAxisType = 2),
						xStart:=T_Process.TFctProcess.xStart ,
						xStop:=T_Process.TFctProcess.xStop ,
						xStopCycle:=T_Process.TFctProcess.xStopCycle,
						xQuitErr:=T_Process.TFctProcess.xQuitErr ,
						xAbord:=T_Process.TFctProcess.xAbord ,
						T_Station:= T_Station,
						T_Process:= T_Process,
						xReset:= xResetAutoGeometry,
						T_ExchgParam:= T_ExchgParam,
						T_NovRAMData:=T_NovRAMData,
						xEnd=>T_Process.TFctProcess.xEnd ,
						xError=>T_Process.TFctProcess.xError ,
						diErrorNr=>T_Process.TFctProcess.diErrorNr);
	xResetAutoGroove:=TRUE;
	FBPrcAutoGroove(	xMicroRodActive:=(T_NovRAMData.T_Standard.T_MachineConfig.iConfigMachineType = 2),
						xBeckhoffDriveActive:=(T_NovRAMData.T_Standard.T_MachineConfig.iConfigAxisType = 2),
						xStart:=T_Process.TFctProcess.xStart ,
						xStop:=T_Process.TFctProcess.xStop ,
						xQuitErr:=T_Process.TFctProcess.xQuitErr ,
						xAbord:=T_Process.TFctProcess.xAbord ,
						T_Station:= T_Station,
						T_Process:= T_Process,
						xReset:= xResetAutoGroove,
						T_ExchgParam:= T_ExchgParam,
						xDoNotMoveGrindPosition:=T_NovRAMData.T_ProcessImageData.T_AutoGroovePara.xBlockGrindFeeder,
						xPlungeActive:=T_NovRAMData.T_ProcessImageData.T_AutoGroovePara.xPlungeActivationGroove,
						T_NovRAMData:=T_NovRAMData,
						xEnd=>T_Process.TFctProcess.xEnd ,
						xError=>T_Process.TFctProcess.xError ,
						diErrorNr=>T_Process.TFctProcess.diErrorNr);
	xResetToolCalibration:=TRUE;
	FBPrcToolCalibration(	xMicroRodActive:=(T_NovRAMData.T_Standard.T_MachineConfig.iConfigMachineType = 2),
						xBeckhoffDriveActive:=(T_NovRAMData.T_Standard.T_MachineConfig.iConfigAxisType = 2),
						xStart:=T_Process.TFctProcess.xStart ,
						xStop:=T_Process.TFctProcess.xStop ,
						xQuitErr:=T_Process.TFctProcess.xQuitErr ,
						xAbord:=T_Process.TFctProcess.xAbord ,
						T_Station:= T_Station,
						T_Process:= T_Process,
						xReset:= xResetToolCalibration,
						T_ExchgParam:= T_ExchgParam,
						T_NovRAMData:=T_NovRAMData,
						xEnd=>T_Process.TFctProcess.xEnd ,
						xError=>T_Process.TFctProcess.xError ,
						diErrorNr=>T_Process.TFctProcess.diErrorNr);
END_IF;
END_FUNCTION_BLOCK

(* POU PRG_PROCESS_LAYER4/FB_PROCESS/FB_PrcMachineReference, ST *)
FUNCTION_BLOCK FB_PrcMachineReference
VAR_INPUT
	xMicroRodActive: BOOL;				(* choice of the machine MicroWire or MicroRod *)
	xBeckhoffDriveActive: BOOL;			(* choice of the axis Beckhoff or EcoStep *)
	T_NovRAMData:ST_DATA_RETAIN;	(* Novram structure for all Machine parameter *)
END_VAR
VAR_IN_OUT
	xStart : BOOL;							(* start a process *)
	xStop : BOOL;							(* stop a process *)
	xQuitErr : BOOL;						(* quit an error *)
	xAbord : BOOL;						(* abord a process *)
	T_Station : ST_STATION;				(* data structure of the stationlevel *)
	T_Process : ST_PROCESS;			(* data strucuture of the processlevel *)
	xReset : BOOL;						(* reset the FB *)
	T_ExchgParam:ST_QVIS_EXCHG_PARAM;	(* data structure of the visualisation *)
END_VAR
VAR_OUTPUT
	xEnd : BOOL;							(* Endflag of the process *)
	xError : BOOL;							(* Errorflag of the process *)
	diErrorNr : DINT;						(* Error number of the process *)
END_VAR
VAR
	iStepPrc: INT;
	xInitStep: BOOL;
	xSetError: BOOL;
	xSetEnd: BOOL;
	xStartMainCtr: BOOL;
	xStartMainPrc: BOOL;
	xInitMainCtr: BOOL;
	xFreeze: BOOL;
	xInitError: BOOL;
	iStepError: INT;
	xTmpStop: BOOL;
	xSetTmpError: BOOL;
	xTmpAbord: BOOL;
	diTmpErrNr: DINT;
	xSetEndPrc : BOOL;
	iTmpFunctionNr:INT;
	xStopFctStation1: BOOL;
	iStepStop: INT;
	iTmpStationFunctionNr: INT;
	xStartProcess: BOOL;
	TONStartTimer: TON;
	tStepTime: TIME;
	TONStartTimer1: TON;
END_VAR
(****************************************************************************************************************************************************)
(***********   This Functionblock define the process for the Machine referencing-->it is needed only for the MicroRod     ************)
(****************************************************************************************************************************************************)

(******************************************************************************************************************************************)
(****************************				           Reset Function Part                                                 *****************************)
(******************************************************************************************************************************************)
IF xReset THEN
	xReset:=FALSE;
	xSetEnd:=TRUE;
END_IF;
(******************************************************************************************************************************************)
(****************************				              Error Controlling Part                                            *****************************)
(******************************************************************************************************************************************)
IF (xSetError OR T_Station.TControl.xError) AND NOT(xSetEnd) THEN
	IF NOT(xInitError) THEN
		iStepError:=100;
		xInitError:=TRUE;
		IF NOT(xSetError) THEN
			xSetError:=TRUE;
			xSetTmpError:=FALSE;
		ELSE
			xSetTmpError:=TRUE;
		END_IF;
	END_IF;
	CASE iStepError OF
		100:	IF T_Station.TControl.xError THEN
				diErrorNr:=T_Station.TControl.diErrorNr;
			END_IF;
			IF xSetTmpError THEN
				diErrorNr:=diTmpErrNr;
			END_IF;
			iStepError:=200;
		200:	IF xSetTmpError THEN
				xSetTmpError:=FALSE;
				xStopFctStation1:=FALSE;
				iStepError:=300;
			ELSE
				IF NOT(T_Station.TControl.xError) AND NOT(T_Station.TControl.xEnd) THEN
					IF (T_Station.TControl.iFunctNr = 1) THEN
						T_Station.TControl.xStop:=TRUE;
						xStopFctStation1:=TRUE;
					ELSE
						xStopFctStation1:=FALSE;
					END_IF;
				END_IF;
				iStepError:=300;
			END_IF;
		300:	IF xStopFctStation1 THEN
				IF NOT(T_Station.TControl.xStop) THEN
					xStopFctStation1:=FALSE;
				END_IF;
			END_IF;
			IF NOT(xStopFctStation1) THEN
				xError:=TRUE;
				iStepError:=400;
			END_IF;
		400:	IF xQuitErr THEN
				T_Station.TControl.xQuitError:=T_Station.TControl.xError;
				iStepError:=500;
			END_IF;
		500: IF NOT(T_Station.TControl.xQuitError) THEN
				xSetEnd:=TRUE;
			END_IF;
	END_CASE;
END_IF;
(******************************************************************************************************************************************)
(****************************				              Main Controlling Part                                            *****************************)
(******************************************************************************************************************************************)
IF (xStart OR xStartMainCtr) AND NOT(xSetEnd) AND NOT(xSetError) THEN
	IF NOT (xInitMainCtr) THEN
		iStepPrc:=10;
		xInitMainCtr:=TRUE;
		xStartMainCtr:=TRUE;
		xStart:=FALSE;
		xEnd:=FALSE;
		xSetEndPrc:=FALSE;
		iTmpFunctionNr:=1;
		xAbord:=FALSE;
	END_IF;
	IF xStop AND NOT(xTmpStop) THEN
		xTmpStop:=TRUE;
		iStepStop:=1;
	END_IF;
	IF xTmpStop THEN
		CASE iStepStop OF
		1:	IF NOT(T_Station.TControl.xEnd) THEN
				T_Station.TControl.xStop:=TRUE;
				iStepStop:=10;
			ELSE
				iStepStop:=20;
			END_IF;
		10:	IF NOT(T_Station.TControl.xStop) THEN
				iStepStop:=20;
			END_IF;
		(* Check Active Movement of the Axis *)
		20:	IF NOT(T_Station.TControl.xStart) AND T_Station.TControl.xEnd THEN
				T_Station.TControl.iFunctNr:=18;	(* Check Axis Movement, and stop it if moves *)
				T_Station.TControl.xStart:=TRUE;
				iStepStop:=30;
			END_IF;
		30:	IF NOT(T_Station.TControl.xStart) AND T_Station.TControl.xEnd THEN
				xStartMainPrc:=FALSE;
				xInitStep:=FALSE;
				iStepPrc:=0;
				xSetEnd:=TRUE;
				RETURN;
			END_IF;
		END_CASE;
		RETURN;
	END_IF;
	IF NOT(xStartMainPrc) THEN
		xStartMainPrc:=TRUE;
	END_IF;
END_IF;
(******************************************************************************************************************************************)
(****************************				             Main Procedure Part                                             *****************************)
(******************************************************************************************************************************************)
IF xStartMainPrc AND NOT(xSetEnd) AND NOT(xSetError) THEN
	CASE iStepPrc OF
		(* Check first if the ToolCalibration is available to start it *)
		10:	T_Station.THardware.TAxisToolLeft.T_CtrleSingle.lrAcceleration:=T_NovRAMData.T_Standard.T_TeachINToolLeft.rAcceleration;
			T_Station.THardware.TAxisToolLeft.T_CtrleSingle.lrDecceleration:=T_NovRAMData.T_Standard.T_TeachINToolLeft.rDeceleration;
			T_Station.THardware.TAxisToolCenter.T_CtrleSingle.lrAcceleration:=T_NovRAMData.T_Standard.T_TeachINToolCenter.rAcceleration;
			T_Station.THardware.TAxisToolCenter.T_CtrleSingle.lrDecceleration:=T_NovRAMData.T_Standard.T_TeachINToolCenter.rDeceleration;
			T_Station.THardware.TAxisToolRight.T_CtrleSingle.lrAcceleration:=T_NovRAMData.T_Standard.T_TeachINToolRight.rAcceleration;
			T_Station.THardware.TAxisToolRight.T_CtrleSingle.lrDecceleration:=T_NovRAMData.T_Standard.T_TeachINToolRight.rDeceleration;
			T_Station.THardware.TAxisToolFeeder.T_CtrleSingle.lrAcceleration:=T_NovRAMData.T_Standard.T_TeachINToolFeeder.rAcceleration;
			T_Station.THardware.TAxisToolFeeder.T_CtrleSingle.lrDecceleration:=T_NovRAMData.T_Standard.T_TeachINToolFeeder.rDeceleration;
			T_Station.THardware.TAxisGrindFeeder.T_CtrleSingle.lrAcceleration:=T_NovRAMData.T_Standard.T_TeachINGrindFeeder.rAcceleration;
			T_Station.THardware.TAxisGrindFeeder.T_CtrleSingle.lrDecceleration:=T_NovRAMData.T_Standard.T_TeachINGrindFeeder.rDeceleration;
			(* On the MicroWire it is not possible to start the Reference Procedure *)
			IF NOT(xMicroRodActive) THEN
				xSetError:=TRUE;
				diTmpErrNr:=5;	(* On the MicroWire it is not possible to Referencing *)
				RETURN;
			END_IF;
			xStartMainPrc:=FALSE;
			xInitStep:=FALSE;
			iStepPrc:=20;
		(* Switch First all Axis the power supply on *)
		20:	IF NOT(xInitStep) THEN
				xInitStep:=TRUE;
				T_Station.TControl.iFunctNr:=16;
				T_Station.TControl.xStart:=TRUE;
			END_IF;
			IF NOT(T_Station.TControl.xStart) AND T_Station.TControl.xEnd THEN
				iStepPrc:=30;
				xStartMainPrc:=FALSE;
				xInitStep:=FALSE;
				iTmpStationFunctionNr:=6;
				T_Station.THardware.TAxisToolLeft.T_CtrleSingle.rSetPosition:=0.0;
				T_Station.THardware.TAxisToolCenter.T_CtrleSingle.rSetPosition:=0.0;
				T_Station.THardware.TAxisToolRight.T_CtrleSingle.rSetPosition:=0.0;
				T_Station.THardware.TAxisToolFeeder.T_CtrleSingle.rSetPosition:=0.0;
			END_IF;
		(* Reset the Position of the Axis *)
		30:	IF NOT(xInitStep) THEN
				xInitStep:=TRUE;
				(* 6=ToolLeft, 7=ToolCenter, 8=ToolRight, 9=ToolFeeder *)
				T_Station.TControl.iFunctNr:=iTmpStationFunctionNr;
				T_Station.TControl.xStart:=TRUE;
			END_IF;
			IF NOT(T_Station.TControl.xStart) AND T_Station.TControl.xEnd THEN
				iTmpStationFunctionNr:=iTmpStationFunctionNr + 1;
				xStartMainPrc:=FALSE;
				xInitStep:=FALSE;
				IF (iTmpStationFunctionNr < 10) THEN
					iStepPrc:=30;
				ELSE
					iStepPrc:=40;
				END_IF;
			END_IF;
		(* GrindFeeder Set Absolut to Security Position *)
		40:	IF NOT(xInitStep) THEN
				xInitStep:=TRUE;
				T_Station.TControl.iFunctNr:=4;
				T_Station.TControl.xStart:=TRUE;
				T_Station.THardware.TAxisGrindFeeder.T_CtrleSingle.lrAcceleration:=T_NovRAMData.T_Standard.T_TeachINGrindFeeder.rAcceleration;
				T_Station.THardware.TAxisGrindFeeder.T_CtrleSingle.lrDecceleration:=T_NovRAMData.T_Standard.T_TeachINGrindFeeder.rDeceleration;
				T_Station.THardware.TAxisGrindFeeder.T_CtrleSingle.lrPosition:=	T_NovRAMData.T_ProcessImageData.T_ProcessPara.rToolDiameterProcess +
																			T_NovRAMData.T_ProcessImageData.T_ProcessPara.rSecurityPosGrindFeedProcess;
				T_Station.THardware.TAxisGrindFeeder.T_CtrleSingle.lrVelocity:=T_NovRAMData.T_ProcessImageData.T_ProcessPara.rSpeedBackwardGrindFeed;
			END_IF;
			IF NOT(T_Station.TControl.xStart) AND T_Station.TControl.xEnd THEN
				iStepPrc:=50;
				xStartMainPrc:=FALSE;
				xInitStep:=FALSE;
			END_IF;
		(* Reference the ToolFeeder *)
		50:	IF NOT(xInitStep) THEN
				xStartProcess:=TRUE;
				xInitStep:=TRUE;
				T_Station.TControl.iFunctNr:=1;
				T_Station.TControl.xStart:=TRUE;
			END_IF;
			IF NOT(T_Station.TControl.xStart) AND T_Station.TControl.xEnd THEN
				xStartMainPrc:=FALSE;
				xInitStep:=FALSE;
				iStepPrc:=60;
			END_IF;
		60:	xSetEndPrc:=FALSE;
			xStartMainPrc:=FALSE;
			xInitStep:=FALSE;
			iStepPrc:=0;
			xSetEnd:=TRUE;
	END_CASE;
END_IF;
(******************************************************************************************************************************************)
(****************************				             	Init / Reset Part                                                   *****************************)
(******************************************************************************************************************************************)
IF xSetEnd THEN
	xEnd:=TRUE;
	xInitStep:=FALSE;
	xSetEnd:=FALSE;
	xStop:=FALSE;
	xStartMainPrc:=FALSE;
	xTmpStop:=FALSE;
	xInitMainCtr:=FALSE;
	xStartMainCtr:=FALSE;
	xStart:=FALSE;
	xSetError:=FALSE;
	xQuitErr:=FALSE;
	xError:=FALSE;
	diErrorNr:=0;
	xInitError:=FALSE;
	xFreeze:=FALSE;
	xAbord:=FALSE;
	xTmpAbord:=FALSE;
	xSetEndPrc:=FALSE;
	xStartProcess:=FALSE;
END_IF;
END_FUNCTION_BLOCK

(* POU PRG_PROCESS_LAYER4/FB_PROCESS/FB_PrcAutoGeometry, ST *)
FUNCTION_BLOCK FB_PrcAutoGeometry
VAR_INPUT
	xMicroRodActive: BOOL;				(* choice of the machine MicroWire or MicroRod *)
	xBeckhoffDriveActive: BOOL;			(* choice of the axis Beckhoff or EcoStep *)
	T_NovRAMData:ST_DATA_RETAIN;	(* Novram structure for all Machine parameter *)
END_VAR
VAR_IN_OUT
	xStart : BOOL;							(* start a process *)
	xStop : BOOL;							(* stop a process *)
	xStopCycle : BOOL;					(* stop a process on the end of the cycle *)
	xQuitErr : BOOL;						(* quit an error *)
	xAbord : BOOL;						(* abord a process *)
	T_Station : ST_STATION;				(* data structure of the stationlevel *)
	T_Process : ST_PROCESS;			(* data strucuture of the processlevel *)
	xReset : BOOL;						(* reset the FB *)
	T_ExchgParam:ST_QVIS_EXCHG_PARAM;	(* data structure of the visualisation *)
END_VAR
VAR_OUTPUT
	xEnd : BOOL;							(* Endflag of the process *)
	xError : BOOL;							(* Errorflag of the process *)
	diErrorNr : DINT;						(* Error number of the process *)
END_VAR
VAR
	iStepPrc: INT;
	xInitStep: BOOL;
	xSetError: BOOL;
	xSetEnd: BOOL;
	xStartMainCtr: BOOL;
	xStartMainPrc: BOOL;
	xInitMainCtr: BOOL;
	xFreeze: BOOL;
	xInitError: BOOL;
	iStepError: INT;
	xTmpStop: BOOL;
	xSetTmpError: BOOL;
	xTmpAbord: BOOL;
	diTmpErrNr: DINT;
	xSetEndPrc : BOOL;
	iTmpFunctionNr:INT;
	xStopFctStation1: BOOL;
	iStepStop: INT;
	FBCheckToolGeometryPara: FB_CheckToolGeometryPara;
	iTmpStationFunctionNr: INT;
	xStartProcess: BOOL;
	TONStartTimer: TON;
	tStepTime: TIME;
	TONStartTimer1: TON;
	xDoNotMovePositionOfToolFeeder: BOOL;
	xTmp: BOOL;
	xTmpStopCycle: BOOL;
	xProcessHold: BOOL;
(*08.07.2014: KFS	{	*)
	TONWarmUpBreakTimer: TON;
	TONWarmUpTimer: TON;
	xWarmUpCycle:BOOL;
	xWarmUp:BOOL;
(*08.07.2014: KFS	}	*)
	xWarmUpDone: BOOL;
END_VAR
(****************************************************************************************************************************************************)
(***********                                      This Functionblock define the process for the AutoGeometry                                                     ************)
(****************************************************************************************************************************************************)

(******************************************************************************************************************************************)
(****************************				           Reset Function Part                                                 *****************************)
(******************************************************************************************************************************************)
IF xReset THEN
	xReset:=FALSE;
	xSetEnd:=TRUE;
END_IF;
(******************************************************************************************************************************************)
(****************************				              Error Controlling Part                                            *****************************)
(******************************************************************************************************************************************)
IF (xSetError OR T_Station.TControl.xError) AND NOT(xSetEnd) THEN
	IF NOT(xInitError) THEN
		iStepError:=100;
		xInitError:=TRUE;
		T_Station.TControl.iCountDownPlungeCycle:=1;
		IF NOT(xSetError) THEN
			xSetError:=TRUE;
			xSetTmpError:=FALSE;
		ELSE
			xSetTmpError:=TRUE;
		END_IF;
	END_IF;
	CASE iStepError OF
		100:	IF T_Station.TControl.xError THEN
				diErrorNr:=T_Station.TControl.diErrorNr;
			END_IF;
			IF xSetTmpError THEN
				diErrorNr:=diTmpErrNr;
			END_IF;
			iStepError:=200;
		200:	IF xSetTmpError THEN
				xSetTmpError:=FALSE;
				xStopFctStation1:=FALSE;
				iStepError:=300;
			ELSE
				IF NOT(T_Station.TControl.xError) AND NOT(T_Station.TControl.xEnd) THEN
					IF (T_Station.TControl.iFunctNr = 1) THEN
						T_Station.TControl.xStop:=TRUE;
						xStopFctStation1:=TRUE;
					ELSE
						xStopFctStation1:=FALSE;
					END_IF;
				END_IF;
				iStepError:=300;
			END_IF;
		300:	IF xStopFctStation1 THEN
				IF NOT(T_Station.TControl.xStop) THEN
					xStopFctStation1:=FALSE;
				END_IF;
			END_IF;
			IF NOT(xStopFctStation1) THEN
				xError:=TRUE;
				iStepError:=400;
			END_IF;
		400:	IF xQuitErr THEN
				T_Station.TControl.xQuitError:=T_Station.TControl.xError;
				iStepError:=500;
			END_IF;
		500: IF NOT(T_Station.TControl.xQuitError) THEN
				xSetEnd:=TRUE;
			END_IF;
	END_CASE;
END_IF;
(******************************************************************************************************************************************)
(****************************				              Main Controlling Part                                            *****************************)
(******************************************************************************************************************************************)
IF (xStart OR xStartMainCtr) AND NOT(xSetEnd) AND NOT(xSetError) THEN
	IF NOT (xInitMainCtr) THEN
		iStepPrc:=10;
		xInitMainCtr:=TRUE;
		xStartMainCtr:=TRUE;
		xStart:=FALSE;
		xEnd:=FALSE;
		xSetEndPrc:=FALSE;
		iTmpFunctionNr:=1;
		xAbord:=FALSE;
		xProcessHold:=FALSE;
		T_ExchgParam.T_InfoValueCommon.iCountDownCycle:=1;
		xDoNotMovePositionOfToolFeeder:=FALSE;
		T_ExchgParam.T_InfoValueCommon.rActualWireFeedPosition:=0.0;
		T_ExchgParam.T_InfoValueCommon.rActualWireFeedSpeed:=0.0;
		(*08.07.2014: KFS	{	*)
		xWarmUp:= xWarmUpCycle:= T_ExchgParam.T_StationCommon.T_AutoGeometryPara.xWarmUp;
		xWarmUpDone:=FALSE;
		(*08.07.2014: KFS	}	*)
	END_IF;
	IF (xStopCycle AND NOT(xTmpStopCycle)) THEN
		IF (T_NovRAMData.T_ProcessImageData.T_AutoGeometryPara.iCycleGeometry <= 1) THEN
			xStopCycle:=xProcessHold:=FALSE;
			RETURN;
		END_IF;
		IF (iStepPrc = 40) AND NOT(xInitStep) THEN
			xTmpStopCycle:=TRUE;
		END_IF;
	END_IF;
	IF xTmpStopCycle THEN
		xStopCycle:=FALSE;
		xProcessHold:=TRUE;
		xTmpStopCycle:=FALSE;
		xInitStep:=xStartMainPrc:=FALSE;
		(*08.07.2014: KFS	{	*)
		xWarmUp:=FALSE;
		(*08.07.2014: KFS	}	*)
		iStepPrc:=100;
		RETURN;
	END_IF;
	IF xStop AND NOT(xTmpStop) THEN
		xTmpStop:=TRUE;
		iStepStop:=1;
	END_IF;
	IF xTmpStop THEN
		CASE iStepStop OF
		1:	IF NOT(T_Station.TControl.xEnd) THEN
				T_Station.TControl.xStop:=TRUE;
				iStepStop:=10;
			ELSE
				iStepStop:=20;
			END_IF;
		10:	IF NOT(T_Station.TControl.xStop) THEN
				iStepStop:=20;
			END_IF;
		20:	IF NOT(T_Station.TControl.xStart) AND T_Station.TControl.xEnd THEN
				T_Station.TControl.iFunctNr:=4;
				T_Station.TControl.xStart:=TRUE;
				T_Station.THardware.TAxisGrindFeeder.T_CtrleSingle.lrAcceleration:=T_NovRAMData.T_Standard.T_TeachINGrindFeeder.rAcceleration;
				T_Station.THardware.TAxisGrindFeeder.T_CtrleSingle.lrDecceleration:=T_NovRAMData.T_Standard.T_TeachINGrindFeeder.rDeceleration;
				T_Station.THardware.TAxisGrindFeeder.T_CtrleSingle.lrPosition:=	T_NovRAMData.T_ProcessImageData.T_ProcessPara.rToolDiameterProcess +
																			T_NovRAMData.T_ProcessImageData.T_ProcessPara.rSecurityPosGrindFeedProcess;
				T_Station.THardware.TAxisGrindFeeder.T_CtrleSingle.lrVelocity:=T_NovRAMData.T_ProcessImageData.T_ProcessPara.rSpeedBackwardGrindFeed;
				iStepStop:=30;
			END_IF;
		(* Check Active Movement of the Axis *)
		30:	IF NOT(T_Station.TControl.xStart) AND T_Station.TControl.xEnd THEN
				T_Station.TControl.iFunctNr:=18;	(* Check Axis Movement, and stop it if moves *)
				T_Station.TControl.xStart:=TRUE;
				iStepStop:=40;
			END_IF;
		40:	IF NOT(T_Station.TControl.xStart) AND T_Station.TControl.xEnd THEN
(*08.07.2014: KFS	{	*)
				IF iStepPrc = 105 THEN
					T_Station.THardware.TCylToolTension.T_CtrleCyl.iFunction:=2;
					T_Station.THardware.TCylToolTension.T_CtrleCyl.T_AnalogCylinder.rForceIn:=T_NovRAMData.T_ProcessImageData.T_ProcessPara.rToolTensionProcess;
					T_Station.THardware.TCylToolTension.T_Config.tDelayOn:=T#1s;
					T_Station.THardware.TCylToolTension.T_CtrleCyl.xExecute:=TRUE;
					T_Station.THardware.TCylToolLeftActive.T_CtrleCyl.iFunction:= 1;
					T_Station.THardware.TCylToolLeftActive.T_CtrleCyl.xExecute:=TRUE;
					T_Station.THardware.TCylToolRightActive.T_CtrleCyl.iFunction:=1;
					T_Station.THardware.TCylToolRightActive.T_CtrleCyl.xExecute:=TRUE;
					T_Station.THardware.TCylToolCenterActive.T_CtrleCyl.iFunction:=1;
					T_Station.THardware.TCylToolCenterActive.T_CtrleCyl.xExecute:=TRUE;
					T_Station.THardware.TCylToolPrismaLeftActive.T_CtrleCyl.iFunction:=1;
					T_Station.THardware.TCylToolPrismaLeftActive.T_CtrleCyl.xExecute:=TRUE;
					T_Station.THardware.TCylToolPrismaRightActive.T_CtrleCyl.iFunction:=1;
					T_Station.THardware.TCylToolPrismaRightActive.T_CtrleCyl.xExecute:=TRUE;
					iStepStop:=45;
				ELSE
(*08.07.2014: KFS	}	*)
					xStartMainPrc:=FALSE;
					xInitStep:=FALSE;
					iStepPrc:=0;
					xSetEnd:=TRUE;
					RETURN;
				END_IF
			END_IF;
		45:IF    (NOT(T_Station.THardware.TCylToolTension.T_CtrleCyl.xExecute) AND T_Station.THardware.TCylToolTension.T_CtrleCyl.xDone ) AND
		             (NOT(T_Station.THardware.TCylToolLeftActive.T_CtrleCyl.xExecute) AND T_Station.THardware.TCylToolLeftActive.T_CtrleCyl.xDone ) AND
			    (NOT(T_Station.THardware.TCylToolRightActive.T_CtrleCyl.xExecute) AND T_Station.THardware.TCylToolRightActive.T_CtrleCyl.xDone ) AND
			    (NOT(T_Station.THardware.TCylToolCenterActive.T_CtrleCyl.xExecute) AND T_Station.THardware.TCylToolCenterActive.T_CtrleCyl.xDone ) AND
			    (NOT(T_Station.THardware.TCylToolPrismaLeftActive.T_CtrleCyl.xExecute) AND T_Station.THardware.TCylToolPrismaLeftActive.T_CtrleCyl.xDone ) AND
			    (NOT(T_Station.THardware.TCylToolPrismaRightActive.T_CtrleCyl.xExecute) AND T_Station.THardware.TCylToolPrismaRightActive.T_CtrleCyl.xDone )		THEN
				xStartMainPrc:=FALSE;
				xInitStep:=FALSE;
				iStepPrc:=0;
				xSetEnd:=TRUE;
				RETURN;
			END_IF;
		END_CASE;
		RETURN;
	END_IF;
	IF NOT(xStartMainPrc) THEN
		xStartMainPrc:=TRUE;
	END_IF;
END_IF;
(******************************************************************************************************************************************)
(****************************				             Main Procedure Part                                             *****************************)
(******************************************************************************************************************************************)
(*08.07.2014: KFS	{	*)
IF xWarmUp AND NOT(xWarmUpDone)THEN
	TONWarmUpTimer(IN:=TRUE,PT:=T#45m);
	IF TONWarmUpTimer.Q THEN
		TONWarmUpTimer(IN:=FALSE);
		xWarmUpDone:=TRUE;
	END_IF;
ELSE
	TONWarmUpTimer(IN:=FALSE);
END_IF;
(*08.07.2014: KFS	}	*)
IF xStartProcess THEN
	TONStartTimer(IN:=TRUE,PT:=T#1s);
	IF TONStartTimer.Q THEN
		TONStartTimer(IN:=FALSE);
		IF (T_ExchgParam.T_InfoValueCommon.tAutoTimeLeft >= T#1s) THEN
			T_ExchgParam.T_InfoValueCommon.tAutoTimeLeft:=T_ExchgParam.T_InfoValueCommon.tAutoTimeLeft - T#1s;
		ELSE
			T_ExchgParam.T_InfoValueCommon.tAutoTimeLeft:=T#0s;
		END_IF;
	END_IF;
	tStepTime:=T_ExchgParam.T_InfoValueCommon.tAutoTimeTotal / 100;
	TONStartTimer1(IN:=TRUE,PT:=tStepTime);
	IF TONStartTimer1.Q THEN
		TONStartTimer1(IN:=FALSE);
		T_ExchgParam.T_InfoValueCommon.bProgressbarAutoGeometry:=T_ExchgParam.T_InfoValueCommon.bProgressbarAutoGeometry + 1;
		IF (T_ExchgParam.T_InfoValueCommon.bProgressbarAutoGeometry >= 100) THEN
			T_ExchgParam.T_InfoValueCommon.bProgressbarAutoGeometry:=100;
		END_IF;
	END_IF;
ELSE
	TONStartTimer(IN:=FALSE);
	TONStartTimer1(IN:=FALSE);
END_IF;
IF xStartMainPrc AND NOT(xSetEnd) AND NOT(xSetError) THEN
	CASE iStepPrc OF
		(* Check first if the AutoGeometry is available to start it *)
		10:	T_Station.THardware.TAxisToolLeft.T_CtrleSingle.lrAcceleration:=T_NovRAMData.T_Standard.T_TeachINToolLeft.rAcceleration;
			T_Station.THardware.TAxisToolLeft.T_CtrleSingle.lrDecceleration:=T_NovRAMData.T_Standard.T_TeachINToolLeft.rDeceleration;
			T_Station.THardware.TAxisToolCenter.T_CtrleSingle.lrAcceleration:=T_NovRAMData.T_Standard.T_TeachINToolCenter.rAcceleration;
			T_Station.THardware.TAxisToolCenter.T_CtrleSingle.lrDecceleration:=T_NovRAMData.T_Standard.T_TeachINToolCenter.rDeceleration;
			T_Station.THardware.TAxisToolRight.T_CtrleSingle.lrAcceleration:=T_NovRAMData.T_Standard.T_TeachINToolRight.rAcceleration;
			T_Station.THardware.TAxisToolRight.T_CtrleSingle.lrDecceleration:=T_NovRAMData.T_Standard.T_TeachINToolRight.rDeceleration;
			T_Station.THardware.TAxisToolFeeder.T_CtrleSingle.lrAcceleration:=T_NovRAMData.T_Standard.T_TeachINToolFeeder.rAcceleration;
			T_Station.THardware.TAxisToolFeeder.T_CtrleSingle.lrDecceleration:=T_NovRAMData.T_Standard.T_TeachINToolFeeder.rDeceleration;
			T_Station.THardware.TAxisGrindFeeder.T_CtrleSingle.lrAcceleration:=T_NovRAMData.T_Standard.T_TeachINGrindFeeder.rAcceleration;
			T_Station.THardware.TAxisGrindFeeder.T_CtrleSingle.lrDecceleration:=T_NovRAMData.T_Standard.T_TeachINGrindFeeder.rDeceleration;
			(* Only for MicroRod, check if the tool is clamped *)
			IF xMicroRodActive THEN
				(*22.12.2009: KFS	{ *)
				(*Added control if all cylinder for the tool are activated*)
				IF ( T_Station.THardware.TCylToolTension.T_CtrleCyl.xStatePosOn AND NOT( xWarmUp) )OR
				    T_Station.THardware.TCylToolLeftActive.T_CtrleCyl.T_Standard.xActivOn OR
 				    T_Station.THardware.TCylToolRightActive.T_CtrleCyl.T_Standard.xActivOn OR
				   (* T_Station.THardware.TCylToolCenterActive.T_CtrleCyl.T_Standard.xActivOn OR*)	(* IGS auskommentiert, diesen Zyl gibts auf der M3 nicht *)
				   ( NOT(T_Station.THardware.TCylToolPrismaLeftActive.T_CtrleCyl.T_Standard.xActivOn) AND NOT(xWarmUp)) OR
				   ( NOT(T_Station.THardware.TCylToolPrismaRightActive.T_CtrleCyl.T_Standard.xActivOn) AND NOT(xWarmUp))  	THEN
						xSetError:=TRUE;
						diTmpErrNr:=2;			(* Tool is not clamped *)
				END_IF;
				(*22.12.2009: KFS	} *)
			END_IF;
			(* Only for MicroRod, check if the Machine is referenced *)
			IF xMicroRodActive THEN
				IF NOT(T_Station.TControl.xReferenced) THEN
					xSetError:=TRUE;
					diTmpErrNr:=1;	(* Machine is not referenced *)
					RETURN;
				END_IF;
			END_IF;
			xStartMainPrc:=FALSE;
			xInitStep:=FALSE;
			iStepPrc:=11;
		(* Set the ToolTension force *)
		11:	IF NOT(xInitStep) THEN
				xInitStep:=TRUE;
				T_Station.THardware.TCylToolTension.T_CtrleCyl.iFunction:=2;	(* activate the ToolTension *)
				T_Station.THardware.TCylToolTension.T_CtrleCyl.T_AnalogCylinder.rForceIn:=T_NovRAMData.T_ProcessImageData.T_ProcessPara.rToolTensionProcess;
				IF xMicroRodActive THEN
					T_Station.THardware.TCylToolTension.T_Config.tDelayOn:=T#1s;
				ELSE
					T_Station.THardware.TCylToolTension.T_Config.tDelayOn:=T#0s;
				END_IF;
				T_Station.THardware.TCylToolTension.T_CtrleCyl.xExecute:=TRUE;
			END_IF;
			IF NOT(T_Station.THardware.TCylToolTension.T_CtrleCyl.xExecute) AND T_Station.THardware.TCylToolTension.T_CtrleCyl.xDone THEN
				(* Only for MicroRod, check if the tool is clamped *)
				IF xMicroRodActive THEN
					IF T_Station.THardware.TCylToolTension.T_CtrleCyl.xStatePosOn AND NOT( xWarmUp) THEN
						xSetError:=TRUE;
						diTmpErrNr:=2;			(* Tool is not clamped *)
						RETURN;
					END_IF;
				END_IF;
				iStepPrc:=20;
				xStartMainPrc:=FALSE;
				xInitStep:=FALSE;
			END_IF;
		(* Switch First all Axis the power supply on *)
		20:	IF NOT(xInitStep) THEN
				xInitStep:=TRUE;
				T_Station.TControl.iFunctNr:=16;
				T_Station.TControl.xStart:=TRUE;
			END_IF;
			IF NOT(T_Station.TControl.xStart) AND T_Station.TControl.xEnd THEN
				iStepPrc:=30;
				xStartMainPrc:=FALSE;
				xInitStep:=FALSE;
				iTmpStationFunctionNr:=6;
				T_Station.THardware.TAxisToolLeft.T_CtrleSingle.rSetPosition:=0.0;
				T_Station.THardware.TAxisToolCenter.T_CtrleSingle.rSetPosition:=0.0;
				T_Station.THardware.TAxisToolRight.T_CtrleSingle.rSetPosition:=0.0;
				T_Station.THardware.TAxisToolFeeder.T_CtrleSingle.rSetPosition:=0.0;
			END_IF;
		(* Reset the Position of the Axis *)
		30:	IF NOT(xInitStep) THEN
				xInitStep:=TRUE;
				(* 6=ToolLeft, 7=ToolCenter, 8=ToolRight, 9=ToolFeeder *)
				T_Station.TControl.iFunctNr:=iTmpStationFunctionNr;
				T_Station.TControl.xStart:=TRUE;
			END_IF;
			IF NOT(T_Station.TControl.xStart) AND T_Station.TControl.xEnd THEN
				iTmpStationFunctionNr:=iTmpStationFunctionNr + 1;
				IF NOT(xMicroRodActive) AND (iTmpStationFunctionNr = 7) THEN
					iTmpStationFunctionNr:=iTmpStationFunctionNr + 1;
				END_IF;
				IF xMicroRodActive AND (iTmpStationFunctionNr = 9) THEN
					iTmpStationFunctionNr:=iTmpStationFunctionNr + 1;
				END_IF;
				xStartMainPrc:=FALSE;
				xInitStep:=FALSE;
				IF (iTmpStationFunctionNr < 10) THEN
					iStepPrc:=30;
				ELSE
					iStepPrc:=40;
				END_IF;
			END_IF;
		(* GrindFeeder Set Absolut to Security Position *)
		40:	IF NOT(xInitStep) THEN
				xInitStep:=TRUE;
				T_Station.TControl.iFunctNr:=4;
				T_Station.TControl.xStart:=TRUE;
				T_Station.THardware.TAxisGrindFeeder.T_CtrleSingle.lrAcceleration:=T_NovRAMData.T_Standard.T_TeachINGrindFeeder.rAcceleration;
				T_Station.THardware.TAxisGrindFeeder.T_CtrleSingle.lrDecceleration:=T_NovRAMData.T_Standard.T_TeachINGrindFeeder.rDeceleration;
				T_Station.THardware.TAxisGrindFeeder.T_CtrleSingle.lrPosition:=	T_NovRAMData.T_ProcessImageData.T_ProcessPara.rToolDiameterProcess +
																			T_NovRAMData.T_ProcessImageData.T_ProcessPara.rSecurityPosGrindFeedProcess;
				T_Station.THardware.TAxisGrindFeeder.T_CtrleSingle.lrVelocity:=T_NovRAMData.T_ProcessImageData.T_ProcessPara.rSpeedBackwardGrindFeed;
			END_IF;
			IF NOT(T_Station.TControl.xStart) AND T_Station.TControl.xEnd THEN
				IF xMicroRodActive THEN
					IF xDoNotMovePositionOfToolFeeder THEN
						iStepPrc:=60;
					ELSE
						iStepPrc:=50;
					END_IF;
				ELSE
					iStepPrc:=60;
				END_IF;
				xStartMainPrc:=FALSE;
				xInitStep:=FALSE;
			END_IF;
		(* Only for MicroRod-->Set ToolFeed Absolut to the Zero Position*)
		50:	IF NOT(xInitStep) THEN
(* 04.04.2011: KFS	{ 	Neu wird die Längeneinstellung des ToolFeeders nicht mehr kontrolliert und direkt auf die StartPos gefahren(vormals RefPos)!
				xInitStep:=TRUE;
				T_Station.TControl.iFunctNr:=14;
				T_Station.TControl.xStart:=TRUE;
				T_Station.THardware.TAxisToolFeeder.T_CtrleSingle.lrAcceleration:=T_NovRAMData.T_Standard.T_TeachINToolFeeder.rAcceleration;
				T_Station.THardware.TAxisToolFeeder.T_CtrleSingle.lrDecceleration:=T_NovRAMData.T_Standard.T_TeachINToolFeeder.rDeceleration;
				T_Station.THardware.TAxisToolFeeder.T_CtrleSingle.lrPosition:=0.0;
				T_Station.THardware.TAxisToolFeeder.T_CtrleSingle.lrVelocity:=T_NovRAMData.T_ProcessImageData.T_ProcessPara.rSpeedStartPosToolFeedProcess;
			END_IF;
			IF NOT(T_Station.TControl.xStart) AND T_Station.TControl.xEnd THEN
 04.04.2011: KFS	}	*)
				(*30.09.2010: KFS	{ *)
				(* Check first settled geometry parameter *)
				FBCheckToolGeometryPara(	iProcessNr:= 1,
											T_GeometryCommon:= T_ExchgParam.T_GeometryCommon,
											T_AutoGeometryPara:= T_NovRAMData.T_ProcessImageData.T_AutoGeometryPara,
											T_AutoGroovePara:= T_NovRAMData.T_ProcessImageData.T_AutoGroovePara,
											T_ProcessPara:= T_NovRamData.T_ProcessImageData.T_ProcessPara,
											rToolDiameter:=T_NovRAMData.T_ProcessImageData.T_ProcessPara.rToolDiameterProcess,
											xMicroRodActive:=xMicroRodActive,
											(*rOffsetMaxToolLength:= T_Station.THardware.TToolFeederWorkLength.T_CtrleCyl.T_Analog.rLengthIn*));
				IF FBCheckToolGeometryPara.xError THEN
					xSetError:=TRUE;
					diTmpErrNr:=FBCheckToolGeometryPara.diErrorNr;
					RETURN;
				END_IF;
				(*30.09.2010: KFS	} *)
				iStepPrc:=55;
				xStartMainPrc:=FALSE;
				xInitStep:=FALSE;
			END_IF;
		(* Only for MicroRod-->Set ToolFeed Absolut to the StartPosition and if more cycle than only the first time *)
		55:	IF NOT(xInitStep) THEN
				xInitStep:=TRUE;
				T_Station.TControl.iFunctNr:=14;
				T_Station.TControl.xStart:=TRUE;
				T_Station.THardware.TAxisToolFeeder.T_CtrleSingle.lrAcceleration:=T_NovRAMData.T_Standard.T_TeachINToolFeeder.rAcceleration;
				T_Station.THardware.TAxisToolFeeder.T_CtrleSingle.lrDecceleration:=T_NovRAMData.T_Standard.T_TeachINToolFeeder.rDeceleration;
				T_Station.THardware.TAxisToolFeeder.T_CtrleSingle.lrPosition:=T_NovRAMData.T_ProcessImageData.T_ProcessPara.rStartPosToolFeedAuto;
				T_Station.THardware.TAxisToolFeeder.T_CtrleSingle.lrVelocity:=T_NovRAMData.T_ProcessImageData.T_ProcessPara.rSpeedStartPosToolFeedProcess;
			END_IF;
			IF NOT(T_Station.TControl.xStart) AND T_Station.TControl.xEnd THEN
				iStepPrc:=60;
				xStartMainPrc:=FALSE;
				xInitStep:=FALSE;
			END_IF;
		(* ToolRotation Start *)
		60:	IF NOT(xInitStep) THEN
				xInitStep:=TRUE;
				T_Station.TControl.iFunctNr:=2;
				T_Station.TControl.xStart:=TRUE;
				(* ToolLeft --> Master *)
				T_Station.THardware.TAxisToolLeft.T_CtrleSingle.lrVelocity:=T_NovRAMData.T_ProcessImageData.T_AutoGeometryPara.rSpeedToolRotationGeometry;
				T_Station.THardware.TAxisToolLeft.T_CtrleSingle.lrAcceleration:=T_NovRAMData.T_Standard.T_TeachINToolLeft.rAcceleration;
				T_Station.THardware.TAxisToolLeft.T_CtrleSingle.lrDecceleration:=T_NovRAMData.T_Standard.T_TeachINToolLeft.rDeceleration;
				IF xMicroRodActive THEN
					(* ToolCenter --> Slave of ToolLeft only by MicroRod *)
					T_Station.THardware.TAxisToolCenter.T_CtrleSingle.lrAcceleration:=T_NovRAMData.T_Standard.T_TeachINToolCenter.rAcceleration;
					T_Station.THardware.TAxisToolCenter.T_CtrleSingle.lrDecceleration:=T_NovRAMData.T_Standard.T_TeachINToolCenter.rDeceleration;
					T_Station.THardware.TAxisToolCenter.T_CtrleSingle.lrGearDivider:=INT_TO_LREAL(T_Station.T_WorkTool.iBaseGearDivider);
					T_Station.THardware.TAxisToolCenter.T_CtrleSingle.lrGearFactor:=(	INT_TO_LREAL(T_Station.T_WorkTool.iBaseGearDivider) /
																					(T_Station.THardware.TAxisToolLeft.T_CtrleSingle.lrGearRatio /
																					T_Station.THardware.TAxisToolCenter.T_CtrleSingle.lrGearRatio)) * -1.0;

					(* ToolRight --> Slave of ToolLeft by MicroWire or Slave of ToolRight by MicroRod *)
					T_Station.THardware.TAxisToolRight.T_CtrleSingle.lrAcceleration:=T_NovRAMData.T_Standard.T_TeachINToolRight.rAcceleration;
					T_Station.THardware.TAxisToolRight.T_CtrleSingle.lrDecceleration:=T_NovRAMData.T_Standard.T_TeachINToolRight.rDeceleration;
					T_Station.THardware.TAxisToolRight.T_CtrleSingle.lrGearDivider:=INT_TO_LREAL(T_Station.T_WorkTool.iBaseGearDivider);
					T_Station.THardware.TAxisToolRight.T_CtrleSingle.lrGearFactor:=	INT_TO_LREAL(T_Station.T_WorkTool.iBaseGearDivider) /
																					(T_Station.THardware.TAxisToolLeft.T_CtrleSingle.lrGearRatio /
		 																			T_Station.THardware.TAxisToolRight.T_CtrleSingle.lrGearRatio);
				END_IF;
				IF NOT(xMicroRodActive) THEN
					(* ToolRight --> Slave of ToolRight by MicroWire *)
					T_Station.THardware.TAxisToolFeeder.T_CtrleSingle.lrAcceleration:=T_NovRAMData.T_Standard.T_TeachINToolFeeder.rAcceleration;
					T_Station.THardware.TAxisToolFeeder.T_CtrleSingle.lrDecceleration:=T_NovRAMData.T_Standard.T_TeachINToolFeeder.rDeceleration;
					T_Station.THardware.TAxisToolFeeder.T_CtrleSingle.lrGearDivider:=INT_TO_LREAL(T_Station.T_WorkTool.iBaseGearDivider);
					T_Station.THardware.TAxisToolFeeder.T_CtrleSingle.lrGearFactor:=	(INT_TO_LREAL(T_Station.T_WorkTool.iBaseGearDivider) /
																					(T_Station.THardware.TAxisToolFeeder.T_CtrleSingle.lrGearRatio /
																					T_Station.THardware.TAxisToolRight.T_CtrleSingle.lrGearRatio)) * -1.0;

					(* ToolRight --> Slave of ToolLeft by MicroWire or Slave of ToolRight by MicroRod *)
					T_Station.THardware.TAxisToolRight.T_CtrleSingle.lrAcceleration:=T_NovRAMData.T_Standard.T_TeachINToolRight.rAcceleration;
					T_Station.THardware.TAxisToolRight.T_CtrleSingle.lrDecceleration:=T_NovRAMData.T_Standard.T_TeachINToolRight.rDeceleration;
					T_Station.THardware.TAxisToolRight.T_CtrleSingle.lrGearDivider:=INT_TO_LREAL(T_Station.T_WorkTool.iBaseGearDivider);
					T_Station.THardware.TAxisToolRight.T_CtrleSingle.lrGearFactor:=	(INT_TO_LREAL(T_Station.T_WorkTool.iBaseGearDivider) /
																					(T_Station.THardware.TAxisToolLeft.T_CtrleSingle.lrGearRatio /
																					T_Station.THardware.TAxisToolRight.T_CtrleSingle.lrGearRatio)) * -1.0;
				END_IF;
			END_IF;
			IF NOT(T_Station.TControl.xStart) AND T_Station.TControl.xEnd THEN
				xStartMainPrc:=FALSE;
				xInitStep:=FALSE;
				iStepPrc:=70;
			END_IF;
		(* GrindFeeder Set Absolut to ToolDiameter minus the offset with the fast speed *)
		70:  	IF NOT(xInitStep) THEN
				xInitStep:=TRUE;
				T_Station.TControl.iFunctNr:=4;
				T_Station.TControl.xStart:=TRUE;
				T_Station.THardware.TAxisGrindFeeder.T_CtrleSingle.lrAcceleration:=T_NovRAMData.T_Standard.T_TeachINGrindFeeder.rAcceleration;
				T_Station.THardware.TAxisGrindFeeder.T_CtrleSingle.lrDecceleration:=T_NovRAMData.T_Standard.T_TeachINGrindFeeder.rDeceleration;
				T_Station.THardware.TAxisGrindFeeder.T_CtrleSingle.lrPosition:=T_NovRAMData.T_ProcessImageData.T_ProcessPara.rToolDiameterProcess + T_NovRAMData.T_ProcessImageData.T_ProcessPara.rOffsetBeforeToolDiaGrindFeedProcess;
				T_Station.THardware.TAxisGrindFeeder.T_CtrleSingle.lrVelocity:=T_NovRAMData.T_ProcessImageData.T_ProcessPara.rSpeedForwardFastGrindFeed;
			END_IF;
			IF NOT(T_Station.TControl.xStart) AND T_Station.TControl.xEnd THEN
				xStartMainPrc:=FALSE;
				xInitStep:=FALSE;
				iStepPrc:=80;
			END_IF;
		(* Working AutoGeometry *)
		80:	IF NOT(xInitStep) THEN
				xStartProcess:=TRUE;
				xInitStep:=TRUE;
				T_Station.TControl.iFunctNr:=19;
				T_Station.TControl.xStart:=TRUE;
			END_IF;
			IF NOT(T_Station.TControl.xStart) AND T_Station.TControl.xEnd THEN
				xStartMainPrc:=FALSE;
				xInitStep:=FALSE;
				iStepPrc:=90;
				RETURN;
			END_IF;
			(* Only for MicroRod, check if the tool is clamped *)
			IF xMicroRodActive THEN
				IF T_Station.THardware.TCylToolTension.T_CtrleCyl.xStatePosOn AND NOT( xWarmUp) THEN
					xStartMainPrc:=FALSE;
					xInitStep:=FALSE;
					iStepPrc:=81;
					RETURN;
				END_IF;
			END_IF;
			T_ExchgParam.T_InfoValueCommon.iCountDownPlungeCycle:=T_Station.TControl.iCountDownPlungeCycle;
		(* Stop the Process, because the Tool is broken *)
		81:	IF NOT(xInitStep) THEN
				xInitStep:=TRUE;
				T_Station.TControl.xStop:=TRUE;
			END_IF;
			IF NOT(T_Station.TControl.xStart) AND T_Station.TControl.xEnd THEN
				xStartMainPrc:=FALSE;
				xInitStep:=FALSE;
				iStepPrc:=82;
			END_IF;
		(* Set the GrindFeeder to the security Position *)
		82:	IF NOT(xInitStep) THEN
				xInitStep:=TRUE;
				T_Station.TControl.iFunctNr:=4;
				T_Station.TControl.xStart:=TRUE;
				T_Station.THardware.TAxisGrindFeeder.T_CtrleSingle.lrAcceleration:=T_NovRAMData.T_Standard.T_TeachINGrindFeeder.rAcceleration;
				T_Station.THardware.TAxisGrindFeeder.T_CtrleSingle.lrDecceleration:=T_NovRAMData.T_Standard.T_TeachINGrindFeeder.rDeceleration;
				T_Station.THardware.TAxisGrindFeeder.T_CtrleSingle.lrPosition:=	T_NovRAMData.T_ProcessImageData.T_ProcessPara.rToolDiameterProcess +
																			T_NovRAMData.T_ProcessImageData.T_ProcessPara.rSecurityPosGrindFeedProcess;
				T_Station.THardware.TAxisGrindFeeder.T_CtrleSingle.lrVelocity:=T_NovRAMData.T_ProcessImageData.T_ProcessPara.rSpeedBackwardGrindFeed;
			END_IF;
			IF NOT(T_Station.TControl.xStart) AND T_Station.TControl.xEnd THEN
				xStartMainPrc:=FALSE;
				xInitStep:=FALSE;
				iStepPrc:=83;
			END_IF;
		(* Check Active Movement of the Axis *)
		83:	IF NOT(xInitStep) THEN
				xInitStep:=TRUE;
				T_Station.TControl.iFunctNr:=18;	(* Check Axis Movement, and stop it if moves *)
				T_Station.TControl.xStart:=TRUE;
			END_IF;
			IF NOT(T_Station.TControl.xStart) AND T_Station.TControl.xEnd THEN
				xSetError:=TRUE;
				diTmpErrNr:=2;			(* Tool is not clamped *)
				RETURN;
			END_IF;
		(* GrindFeeder Set Absolut to Security Position *)
		90:	IF NOT(xInitStep) THEN
				xInitStep:=TRUE;
				T_Station.TControl.iFunctNr:=4;
				T_Station.TControl.xStart:=TRUE;
				T_Station.THardware.TAxisGrindFeeder.T_CtrleSingle.lrAcceleration:=T_NovRAMData.T_Standard.T_TeachINGrindFeeder.rAcceleration;
				T_Station.THardware.TAxisGrindFeeder.T_CtrleSingle.lrDecceleration:=T_NovRAMData.T_Standard.T_TeachINGrindFeeder.rDeceleration;
				T_Station.THardware.TAxisGrindFeeder.T_CtrleSingle.lrPosition:=	T_NovRAMData.T_ProcessImageData.T_ProcessPara.rToolDiameterProcess +
																			T_NovRAMData.T_ProcessImageData.T_ProcessPara.rSecurityPosGrindFeedProcess;
				T_Station.THardware.TAxisGrindFeeder.T_CtrleSingle.lrVelocity:=T_NovRAMData.T_ProcessImageData.T_ProcessPara.rSpeedBackwardGrindFeed;
			END_IF;
			IF NOT(T_Station.TControl.xStart) AND T_Station.TControl.xEnd THEN
				xStartMainPrc:=FALSE;
				xInitStep:=FALSE;
				IF (T_NovRAMData.T_ProcessImageData.T_AutoGeometryPara.iCycleGeometry > T_ExchgParam.T_InfoValueCommon.iCountDownCycle) THEN
					IF NOT(xStopCycle) THEN
						T_ExchgParam.T_InfoValueCommon.iCountDownCycle:=T_ExchgParam.T_InfoValueCommon.iCountDownCycle + 1;
					END_IF;
					xDoNotMovePositionOfToolFeeder:=TRUE;
					iStepPrc:=40;	(* Repeat to work the same Geometry *)
				ELSE
					iStepPrc:=100;
				END_IF;
			END_IF;
		(* ToolRotation Stop *)
		100:	IF NOT(xInitStep) THEN
				xInitStep:=TRUE;
				T_Station.TControl.iFunctNr:=3;
				T_Station.TControl.xStart:=TRUE;
				(* ToolLeft --> Master *)
				T_Station.THardware.TAxisToolLeft.T_CtrleSingle.lrAcceleration:=T_NovRAMData.T_Standard.T_TeachINToolLeft.rAcceleration;
				T_Station.THardware.TAxisToolLeft.T_CtrleSingle.lrDecceleration:=T_NovRAMData.T_Standard.T_TeachINToolLeft.rDeceleration;
				IF xMicroRodActive THEN
					(* ToolCenter --> Slave of ToolLeft only by MicroRod *)
					T_Station.THardware.TAxisToolCenter.T_CtrleSingle.lrAcceleration:=T_NovRAMData.T_Standard.T_TeachINToolCenter.rAcceleration;
					T_Station.THardware.TAxisToolCenter.T_CtrleSingle.lrDecceleration:=T_NovRAMData.T_Standard.T_TeachINToolCenter.rDeceleration;
				END_IF;
				(* ToolRight --> Slave of ToolLeft by MicroWire or Slave of ToolRight by MicroRod *)
				T_Station.THardware.TAxisToolRight.T_CtrleSingle.lrAcceleration:=T_NovRAMData.T_Standard.T_TeachINToolRight.rAcceleration;
				T_Station.THardware.TAxisToolRight.T_CtrleSingle.lrDecceleration:=T_NovRAMData.T_Standard.T_TeachINToolRight.rDeceleration;
				IF NOT(xMicroRodActive) THEN
					(* ToolRight --> Slave of ToolRight by MicroWire *)
					T_Station.THardware.TAxisToolFeeder.T_CtrleSingle.lrAcceleration:=T_NovRAMData.T_Standard.T_TeachINToolFeeder.rAcceleration;
					T_Station.THardware.TAxisToolFeeder.T_CtrleSingle.lrDecceleration:=T_NovRAMData.T_Standard.T_TeachINToolFeeder.rDeceleration;
				END_IF;
			END_IF;
			IF NOT(T_Station.TControl.xStart) AND T_Station.TControl.xEnd THEN
				xStartMainPrc:=FALSE;
				xInitStep:=FALSE;
				IF NOT(xWarmUpCycle) THEN
					iStepPrc:=110;
				ELSE
					iStepPrc:=102;
				END_IF;
			END_IF;
(*08.07.2014: KFS	{	*)
		102:	IF NOT(xInitStep) THEN
				T_Station.THardware.TCylToolTension.T_CtrleCyl.iFunction:=1;
				T_Station.THardware.TCylToolTension.T_CtrleCyl.xExecute:=TRUE;
				T_Station.THardware.TCylToolLeftActive.T_CtrleCyl.iFunction:= 2;
				T_Station.THardware.TCylToolLeftActive.T_CtrleCyl.xExecute:=TRUE;
				T_Station.THardware.TCylToolRightActive.T_CtrleCyl.iFunction:=2;
				T_Station.THardware.TCylToolRightActive.T_CtrleCyl.xExecute:=TRUE;
				T_Station.THardware.TCylToolCenterActive.T_CtrleCyl.iFunction:=2;
				T_Station.THardware.TCylToolCenterActive.T_CtrleCyl.xExecute:=TRUE;
				T_Station.THardware.TCylToolPrismaLeftActive.T_CtrleCyl.iFunction:=51;
				T_Station.THardware.TCylToolPrismaLeftActive.T_CtrleCyl.xExecute:=TRUE;
				T_Station.THardware.TCylToolPrismaRightActive.T_CtrleCyl.iFunction:=51;
				T_Station.THardware.TCylToolPrismaRightActive.T_CtrleCyl.xExecute:=TRUE;
				xInitStep:=TRUE;
			END_IF;
			IF(NOT(T_Station.THardware.TCylToolTension.T_CtrleCyl.xExecute) AND T_Station.THardware.TCylToolTension.T_CtrleCyl.xDone ) AND
			    (NOT(T_Station.THardware.TCylToolLeftActive.T_CtrleCyl.xExecute) AND T_Station.THardware.TCylToolLeftActive.T_CtrleCyl.xDone ) AND
			    (NOT(T_Station.THardware.TCylToolRightActive.T_CtrleCyl.xExecute) AND T_Station.THardware.TCylToolRightActive.T_CtrleCyl.xDone ) AND
			    (NOT(T_Station.THardware.TCylToolCenterActive.T_CtrleCyl.xExecute) AND T_Station.THardware.TCylToolCenterActive.T_CtrleCyl.xDone ) AND
			    (NOT(T_Station.THardware.TCylToolPrismaLeftActive.T_CtrleCyl.xExecute) AND T_Station.THardware.TCylToolPrismaLeftActive.T_CtrleCyl.xDone ) AND
			    (NOT(T_Station.THardware.TCylToolPrismaRightActive.T_CtrleCyl.xExecute) AND T_Station.THardware.TCylToolPrismaRightActive.T_CtrleCyl.xDone )		THEN
				TONWarmUpBreakTimer(IN:=FALSE);
				xStartMainPrc:=FALSE;
				xInitStep:=FALSE;
				iStepPrc:=105;
			END_IF;
		105: IF xWarmUpDone THEN
				T_ExchgParam.T_StationCommon.T_AutoGeometryPara.xWarmUp:=FALSE;
			END_IF;
			TONWarmUpBreakTimer(IN:=TRUE,PT:=T#20s);
			IF TONWarmUpBreakTimer.Q THEN
				TONWarmUpBreakTimer(IN:=FALSE);
				T_ExchgParam.T_InfoValueCommon.iCountDownCycle:=1;
				xDoNotMovePositionOfToolFeeder:=FALSE;
				xStartMainPrc:=FALSE;
				xInitStep:=FALSE;
				iStepPrc:=107;
			END_IF;
		107:	IF NOT(xInitStep) THEN
				T_Station.THardware.TCylToolTension.T_CtrleCyl.iFunction:=2;
				T_Station.THardware.TCylToolTension.T_CtrleCyl.T_AnalogCylinder.rForceIn:=T_NovRAMData.T_ProcessImageData.T_ProcessPara.rToolTensionProcess;
				T_Station.THardware.TCylToolTension.T_Config.tDelayOn:=T#1s;
				T_Station.THardware.TCylToolTension.T_CtrleCyl.xExecute:=TRUE;
				T_Station.THardware.TCylToolLeftActive.T_CtrleCyl.iFunction:= 1;
				T_Station.THardware.TCylToolLeftActive.T_CtrleCyl.xExecute:=TRUE;
				T_Station.THardware.TCylToolRightActive.T_CtrleCyl.iFunction:=1;
				T_Station.THardware.TCylToolRightActive.T_CtrleCyl.xExecute:=TRUE;
				T_Station.THardware.TCylToolCenterActive.T_CtrleCyl.iFunction:=1;
				T_Station.THardware.TCylToolCenterActive.T_CtrleCyl.xExecute:=TRUE;
				T_Station.THardware.TCylToolPrismaLeftActive.T_CtrleCyl.iFunction:=51;
				T_Station.THardware.TCylToolPrismaLeftActive.T_CtrleCyl.xExecute:=TRUE;
				T_Station.THardware.TCylToolPrismaRightActive.T_CtrleCyl.iFunction:=51;
				T_Station.THardware.TCylToolPrismaRightActive.T_CtrleCyl.xExecute:=TRUE;
				xInitStep:=TRUE;
			END_IF;
			IF(NOT(T_Station.THardware.TCylToolTension.T_CtrleCyl.xExecute) AND T_Station.THardware.TCylToolTension.T_CtrleCyl.xDone ) AND
			    (NOT(T_Station.THardware.TCylToolLeftActive.T_CtrleCyl.xExecute) AND T_Station.THardware.TCylToolLeftActive.T_CtrleCyl.xDone ) AND
			    (NOT(T_Station.THardware.TCylToolRightActive.T_CtrleCyl.xExecute) AND T_Station.THardware.TCylToolRightActive.T_CtrleCyl.xDone ) AND
			    (NOT(T_Station.THardware.TCylToolCenterActive.T_CtrleCyl.xExecute) AND T_Station.THardware.TCylToolCenterActive.T_CtrleCyl.xDone ) AND
			    (NOT(T_Station.THardware.TCylToolPrismaLeftActive.T_CtrleCyl.xExecute) AND T_Station.THardware.TCylToolPrismaLeftActive.T_CtrleCyl.xDone ) AND
			    (NOT(T_Station.THardware.TCylToolPrismaRightActive.T_CtrleCyl.xExecute) AND T_Station.THardware.TCylToolPrismaRightActive.T_CtrleCyl.xDone )		THEN
				xStartMainPrc:=FALSE;
				xInitStep:=FALSE;
				iStepPrc:=10;
			END_IF;
(*08.07.2014: KFS	}	*)
		110:	xSetEndPrc:=FALSE;
			xStartMainPrc:=FALSE;
			xInitStep:=FALSE;
			iStepPrc:=0;
			xSetEnd:=TRUE;
	END_CASE;
END_IF;
(******************************************************************************************************************************************)
(****************************				             	Init / Reset Part                                                   *****************************)
(******************************************************************************************************************************************)
IF xSetEnd THEN
	xEnd:=TRUE;
	xInitStep:=FALSE;
	xSetEnd:=FALSE;
	xStop:=FALSE;
	xStopCycle:=FALSE;
	xTmpStopCycle:=FALSE;
	xStartMainPrc:=FALSE;
	xTmpStop:=FALSE;
	xInitMainCtr:=FALSE;
	xStartMainCtr:=FALSE;
	xStart:=FALSE;
	xSetError:=FALSE;
	xQuitErr:=FALSE;
	xError:=FALSE;
	diErrorNr:=0;
	xInitError:=FALSE;
	xFreeze:=FALSE;
	xAbord:=FALSE;
	xTmpAbord:=FALSE;
	xSetEndPrc:=FALSE;
	xStartProcess:=FALSE;
(*08.07.2014: KFS	{	*)
	xWarmUp:= xWarmUpCycle:= FALSE;
	xWarmUpDone:=FALSE;
(*08.07.2014: KFS	}	*)
END_IF;
END_FUNCTION_BLOCK

(* POU GENERAL/FB_CheckToolGeometryPara, ST *)
FUNCTION_BLOCK FB_CheckToolGeometryPara
VAR_INPUT
	iProcessNr:INT;	(* 1=AutoGeometry, 2=AutoGroove *)
	T_GeometryCommon:ST_GEOMETRY_COMMON;
	T_AutoGeometryPara:ST_EXCHG_PARAM_AUTOGEOMETRY;
	T_AutoGroovePara:ST_EXCHG_PARAM_AUTOGROOVE;
	T_ProcessPara:ST_EXCHG_PARAM_PROCESS;
	rToolDiameter:REAL;
(*22.12.2009: KFS 	{    *)
	xMicroRodActive: BOOL;				(* choice of the machine MicroWire or MicroRod *)
(*04.04.2011: KFS	{
	rOffsetMaxToolLength:REAL;
04.04.2011: KFS	}   *)
(*22.12.2009: KFS 	}   *)
END_VAR
VAR_OUTPUT
	xError:BOOL;		(* errorflag *)
	diErrorNr: DINT;	(* number of the caused error *)
(*22.12.2009: KFS 	{    *)
	xMultiCycleGrindFeedGeometry: BOOL;				(* choice of multicycle for MicroRod *)
(*22.12.2009: KFS 	}   *)
END_VAR
VAR
	ii: INT;
	rToolLength: REAL;
	rToolDiamterMax: REAL;
	rToolDiamterMin: REAL;
END_VAR
(****************************************************************************************************************************************************)
(***********                         check the settled value of the geometry and set an error if the value ar not correct                         ************)
(****************************************************************************************************************************************************)
(* Check ToolLength *)
	rToolLength:=0;
	diErrorNr:=0;
	xError:=FALSE;
	xMultiCycleGrindFeedGeometry:= FALSE;
	FOR ii:=1 TO 4 DO
		IF T_GeometryCommon.T_Geometry.axActiveSection[ii] THEN
			rToolLength:=rToolLength + T_GeometryCommon.T_Geometry.arSectionLength[ii];
		END_IF;
	END_FOR;
(*
	IF (iProcessNr = 1) THEN
		IF T_AutoGeometryPara.xPlungeActivationGeometry THEN
			rToolLength:=rToolLength + (T_AutoGeometryPara.rPlungeLengthToolFeedGeometry / 10.0);
		END_IF;
		IF T_AutoGeometryPara.xDisplaceActivationGeometry THEN
			rToolLength:=rToolLength + (T_AutoGeometryPara.rDisplaceLengthToolFeedGeometry / 10.0);
		END_IF;
		IF (T_AutoGeometryPara.iCycleGeometry > 1) THEN
			rToolLength:=rToolLength * INT_TO_REAL(T_AutoGeometryPara.iCycleGeometry);
		END_IF;
	END_IF;
	IF (iProcessNr = 2) THEN
		IF T_AutoGroovePara.xPlungeActivationGroove THEN
			rToolLength:=rToolLength + (T_AutoGroovePara.rPlungeLengthToolFeedGroove / 10.0);
		END_IF;
		IF T_AutoGroovePara.xDisplaceActivationGroove THEN
			rToolLength:=rToolLength + (T_AutoGroovePara.rDisplaceLengthToolFeedGroove / 10.0);
		END_IF;
	END_IF;
*)
	(*22.12.2009: KFS 	{    *)
	IF xMicroRodActive THEN
		IF rToolLength > (T_GeometryCommon.rMaxToolLength - T_ProcessPara.rStartPosToolFeedAuto * 0.1(* - rOffsetMaxToolLength*) ) THEN
			diErrorNr:=16#F201;	(* Settled parameter for ToolLength is to long *)
		END_IF;
		IF rToolLength < T_GeometryCommon.rMinToolLength THEN
			diErrorNr:=16#F202;	(* Settled parameter for ToolLength is to short *)
		END_IF;
	ELSE
		IF rToolLength > T_GeometryCommon.rMaxToolLength THEN
			diErrorNr:=16#F201;	(* Settled parameter for ToolLength is to long *)
		END_IF;
		IF rToolLength < T_GeometryCommon.rMinToolLength THEN
			diErrorNr:=16#F202;	(* Settled parameter for ToolLength is to short *)
		END_IF;
	END_IF;
	(*22.12.2009: KFS	}   *)
(* Check ToolDiamter in case of the prisma *)
	rToolDiamterMax:=0;
	FOR ii:=1 TO 4 DO
		IF T_GeometryCommon.T_Geometry.axActiveSection[ii] THEN
			IF (T_GeometryCommon.T_Geometry.arStartDiameter[ii] > rToolDiamterMax) THEN
				rToolDiamterMax:=T_GeometryCommon.T_Geometry.arStartDiameter[ii];
			END_IF;
			IF (T_GeometryCommon.T_Geometry.arEndDiameter[ii] > rToolDiamterMax) THEN
				rToolDiamterMax:=T_GeometryCommon.T_Geometry.arEndDiameter[ii];
			END_IF;
		END_IF;
	END_FOR;
	rToolDiamterMin:=999999;
	FOR ii:=1 TO 4 DO
		IF T_GeometryCommon.T_Geometry.axActiveSection[ii] THEN
			IF (T_GeometryCommon.T_Geometry.arStartDiameter[ii] < rToolDiamterMin) THEN
				rToolDiamterMin:=T_GeometryCommon.T_Geometry.arStartDiameter[ii];
			END_IF;
			IF (T_GeometryCommon.T_Geometry.arEndDiameter[ii] < rToolDiamterMin) THEN
				rToolDiamterMin:=T_GeometryCommon.T_Geometry.arEndDiameter[ii];
			END_IF;
		END_IF;
	END_FOR;
	IF (rToolDiamterMax > T_GeometryCommon.rMaxToolDiameter) THEN
		diErrorNr:=16#F203;	(* Settled parameter for ToolDiameter is to big *)
	END_IF;
	IF (rToolDiamterMin < T_GeometryCommon.rMinToolDiameter) THEN
		diErrorNr:=16#F204;	(* Settled parameter for ToolDiameter is to small *)
	END_IF;
	(*22.12.2009: KFS 	{    *)
(* Check activation for multicycle of the AutoGeometry *)
	IF xMicroRodActive THEN
		IF ( (rToolDiameter - rToolDiamterMin) > T_AutoGeometryPara.rPlungeCycleGrindFeedGeometry ) THEN
			xMultiCycleGrindFeedGeometry := TRUE;
		END_IF;
	END_IF;
	(*22.12.2009: KFS 	}    *)
(* Check the passage from one section to another section if equal *)
	FOR ii:=1 TO 4 DO
		IF T_GeometryCommon.T_Geometry.axActiveSection[ii] THEN
			IF (ii < 4) THEN
				IF T_GeometryCommon.T_Geometry.axActiveSection[ii+ 1] THEN
					IF (T_GeometryCommon.T_Geometry.arEndDiameter[ii] <> T_GeometryCommon.T_Geometry.arStartDiameter[ii + 1]) THEN
						diErrorNr:=16#F205;	(* At least a passage of a section is not equal *)
					END_IF;
				END_IF;
			END_IF;
		END_IF;
	END_FOR;
(* Check ToolDiamter in case of the settled ToolDiameter *)
	rToolDiamterMax:=0;
	FOR ii:=1 TO 4 DO
		IF T_GeometryCommon.T_Geometry.axActiveSection[ii] THEN
			IF (T_GeometryCommon.T_Geometry.arStartDiameter[ii] > rToolDiamterMax) THEN
				rToolDiamterMax:=T_GeometryCommon.T_Geometry.arStartDiameter[ii];
			END_IF;
			IF (T_GeometryCommon.T_Geometry.arEndDiameter[ii] > rToolDiamterMax) THEN
				rToolDiamterMax:=T_GeometryCommon.T_Geometry.arEndDiameter[ii];
			END_IF;
		END_IF;
	END_FOR;
	IF (rToolDiamterMax > rToolDiameter) THEN
		diErrorNr:=16#F206;	(* At least one settled diameter is bigger than the ToolDiameter *)
	END_IF;
	IF (diErrorNr <> 0) THEN
		xError:=TRUE;
	END_IF;
END_FUNCTION_BLOCK

(* POU PRG_PROCESS_LAYER4/FB_PROCESS/FB_PrcAutoGroove, ST *)
FUNCTION_BLOCK FB_PrcAutoGroove
VAR_INPUT
	xMicroRodActive: BOOL;				(* choice of the machine MicroWire or MicroRod *)
	xBeckhoffDriveActive: BOOL;			(* choice of the axis Beckhoff or EcoStep *)
	T_NovRAMData:ST_DATA_RETAIN;	(* Novram structure for all Machine parameter *)
END_VAR
VAR_IN_OUT
	xStart : BOOL;							(* start a process *)
	xStop : BOOL;							(* stop a process *)
	xQuitErr : BOOL;						(* quit an error *)
	xAbord : BOOL;						(* abord a process *)
	T_Station : ST_STATION;				(* data structure of the stationlevel *)
	T_Process : ST_PROCESS;			(* data strucuture of the processlevel *)
	xReset : BOOL;						(* reset the FB *)
	T_ExchgParam:ST_QVIS_EXCHG_PARAM;	(* data structure of the visualisation *)
	xDoNotMoveGrindPosition:BOOL;		(* choice of the AutoGroove process, TRUE=override the GrindAxis position with the ToolDiameter, FALSE=no overriding *)
	xPlungeActive:BOOL;					(* TRUE=Plunge on AutoGroove active, FALSE=Plunge on AutoGroove deactivatet *)
END_VAR
VAR_OUTPUT
	xEnd : BOOL;							(* Endflag of the process *)
	xError : BOOL;							(* Errorflag of the process *)
	diErrorNr : DINT;						(* Error number of the process *)
END_VAR
VAR
	iStepPrc: INT;
	xInitStep: BOOL;
	xSetError: BOOL;
	xSetEnd: BOOL;
	xStartMainCtr: BOOL;
	xStartMainPrc: BOOL;
	xInitMainCtr: BOOL;
	xFreeze: BOOL;
	xInitError: BOOL;
	iStepError: INT;
	xTmpStop: BOOL;
	xSetTmpError: BOOL;
	xTmpAbord: BOOL;
	diTmpErrNr: DINT;
	xSetEndPrc : BOOL;
	iTmpFunctionNr:INT;
	xStopFctStation1: BOOL;
	iStepStop: INT;
	FBCheckToolGeometryPara: FB_CheckToolGeometryPara;
	iTmpStationFunctionNr: INT;
	xStartProcess: BOOL;
	TONStartTimer: TON;
	tStepTime: TIME;
	TONStartTimer1: TON;
	rCheckStartPosition: REAL;
	(*22.12.2009: KFS	{ *)
	iNumberOfGrooves: INT;
	lrAxisToolLeftActuelPosition: LREAL;
	rStartPosAutoGrooveToolRotation: LREAL;
	rOffsetStartPositionGrooves: REAL;
	xOneTimeCheckGeometry:BOOL;
	(*22.12.2009: KFS	} *)
	rMaxTol: REAL:= 5.0;
	xNotFirstGrooveCycle: BOOL;
END_VAR
(****************************************************************************************************************************************************)
(***********                                      This Functionblock define the process for the AutoGroove                                                         ************)
(****************************************************************************************************************************************************)

